LIN {X 0,Y 559.913,Z 737.575,A -85,B 0,C 180,E1 26462.456,E2 26462.456} C_VEL
LIN {X 0,Y 559.908,Z 738.885,A -85,B 0,C 180,E1 26460.511,E2 26460.511} C_VEL
LIN {X 0,Y 559.912,Z 738.467,A -85,B 0,C 180,E1 26458.465,E2 26458.465} C_VEL
LIN {X 0,Y 559.91,Z 736.338,A -85,B 0,C 180,E1 26456.519,E2 26456.519} C_VEL
LIN {X 0,Y 559.924,Z 732.455,A -85,B 0,C 180,E1 26454.569,E2 26454.569} C_VEL
LIN {X 0,Y 559.957,Z 726.723,A -85,B 0,C 180,E1 26452.613,E2 26452.613} C_VEL
LIN {X 0,Y 560.036,Z 718.997,A -85,B 0,C 180,E1 26450.649,E2 26450.649} C_VEL
LIN {X 0,Y 560.157,Z 709.621,A -85,B 0,C 180,E1 26448.781,E2 26448.781} C_VEL
LIN {X 0,Y 560.34,Z 698.616,A -85,B 0,C 180,E1 26447.007,E2 26447.007} C_VEL
LIN {X 0,Y 560.569,Z 686.811,A -85,B 0,C 180,E1 26445.434,E2 26445.434} C_VEL
LIN {X 0,Y 560.869,Z 673.245,A -85,B 0,C 180,E1 26443.921,E2 26443.921} C_VEL
LIN {X 0,Y 561.22,Z 658.578,A -85,B 0,C 180,E1 26442.549,E2 26442.549} C_VEL
LIN {X 0,Y 561.616,Z 642.337,A -85,B 0,C 180,E1 26441.287,E2 26441.287} C_VEL
LIN {X 0,Y 562.015,Z 624.834,A -85,B 0,C 180,E1 26440.178,E2 26440.178} C_VEL
LIN {X 0,Y 561.226,Z 618.186,A -85,B 0,C 180,E1 26439.775,E2 26439.775} C_VEL
LIN {X 0,Y 555.927,Z 601.44,A -85,B 0,C 180,E1 26438.77,E2 26438.77} C_VEL
LIN {X 0,Y 555.124,Z 594.384,A -85,B 0,C 180,E1 26438.452,E2 26438.452} C_VEL
LIN {X 0,Y 555.482,Z 575.161,A -85,B 0,C 180,E1 26437.832,E2 26437.832} C_VEL
LIN {X 0,Y 555.742,Z 555.75,A -85,B 0,C 180,E1 26437.414,E2 26437.414} C_VEL
LIN {X 0,Y 556.621,Z 349.619,A -85,B 0,C 180,E1 26434.588,E2 26434.588} C_VEL
LIN {X 0,Y 555.366,Z 342.045,A -85,B 0,C 180,E1 26434.399,E2 26434.399} C_VEL
LIN {X 0,Y 556.271,Z 299.379,A -85,B 0,C 180,E1 26431.026,E2 26431.026} C_VEL
LIN {X 0,Y 556.522,Z 280.46,A -85,B 0,C 180,E1 26429.484,E2 26429.484} C_VEL
LIN {X 0,Y 552.328,Z 267.902,A -85,B 0,C 180,E1 26428.132,E2 26428.132} C_VEL
LIN {X 0,Y 552.336,Z 267.663,A -85,B 0,C 180,E1 26425.089,E2 26425.089} C_VEL
LIN {X 0,Y 552.305,Z 267.685,A -85,B 0,C 180,E1 26421.746,E2 26421.746} C_VEL
LIN {X 0,Y 552.329,Z 267.679,A -85,B 0,C 180,E1 26418.366,E2 26418.366} C_VEL
LIN {X 0,Y 552.339,Z 267.686,A -85,B 0,C 180,E1 26415.057,E2 26415.057} C_VEL
LIN {X 0,Y 552.324,Z 267.684,A -85,B 0,C 180,E1 26411.768,E2 26411.768} C_VEL
LIN {X 0,Y 552.343,Z 267.678,A -85,B 0,C 180,E1 26408.383,E2 26408.383} C_VEL
LIN {X 0,Y 552.324,Z 267.683,A -85,B 0,C 180,E1 26405.02,E2 26405.02} C_VEL
LIN {X 0,Y 552.341,Z 267.686,A -85,B 0,C 180,E1 26401.667,E2 26401.667} C_VEL
LIN {X 0,Y 552.342,Z 267.677,A -85,B 0,C 180,E1 26398.313,E2 26398.313} C_VEL
LIN {X 0,Y 552.304,Z 267.68,A -85,B 0,C 180,E1 26394.95,E2 26394.95} C_VEL
LIN {X 0,Y 552.333,Z 267.683,A -85,B 0,C 180,E1 26391.673,E2 26391.673} C_VEL
LIN {X 0,Y 552.325,Z 267.683,A -85,B 0,C 180,E1 26388.361,E2 26388.361} C_VEL
LIN {X 0,Y 552.28,Z 267.68,A -85,B 0,C 180,E1 26385.113,E2 26385.113} C_VEL
LIN {X 0,Y 552.331,Z 267.688,A -85,B 0,C 180,E1 26381.911,E2 26381.911} C_VEL
LIN {X 0,Y 552.275,Z 267.688,A -85,B 0,C 180,E1 26378.695,E2 26378.695} C_VEL
LIN {X 0,Y 552.348,Z 268.019,A -85,B 0,C 180,E1 26378.406,E2 26378.406} C_VEL
LIN {X 0,Y 555.682,Z 279.748,A -85,B 0,C 180,E1 26377.289,E2 26377.289} C_VEL
LIN {X 0,Y 555.546,Z 319.159,A -85,B 0,C 180,E1 26374.233,E2 26374.233} C_VEL
LIN {X 0,Y 555.163,Z 359.793,A -85,B 0,C 180,E1 26371.085,E2 26371.085} C_VEL
LIN {X 0,Y 554.627,Z 395.794,A -85,B 0,C 180,E1 26368.297,E2 26368.297} C_VEL
LIN {X 0,Y 553.969,Z 440.023,A -85,B 0,C 180,E1 26364.875,E2 26364.875} C_VEL
LIN {X 0,Y 553.523,Z 472.352,A -85,B 0,C 180,E1 26362.411,E2 26362.411} C_VEL
LIN {X 0,Y 554.186,Z 480.588,A -85,B 0,C 180,E1 26362.264,E2 26362.264} C_VEL
LIN {X 0,Y 553.701,Z 615.423,A -85,B 0,C 180,E1 26360.465,E2 26360.465} C_VEL
LIN {X 0,Y 553.549,Z 631.717,A -85,B 0,C 180,E1 26360.048,E2 26360.048} C_VEL
LIN {X 0,Y 553.324,Z 647.903,A -85,B 0,C 180,E1 26359.427,E2 26359.427} C_VEL
LIN {X 0,Y 553.052,Z 662.877,A -85,B 0,C 180,E1 26358.636,E2 26358.636} C_VEL
LIN {X 0,Y 552.78,Z 676.977,A -85,B 0,C 180,E1 26357.678,E2 26357.678} C_VEL
LIN {X 0,Y 552.532,Z 689.984,A -85,B 0,C 180,E1 26356.555,E2 26356.555} C_VEL
LIN {X 0,Y 552.317,Z 701.515,A -85,B 0,C 180,E1 26355.32,E2 26355.32} C_VEL
LIN {X 0,Y 552.148,Z 711.975,A -85,B 0,C 180,E1 26353.917,E2 26353.917} C_VEL
LIN {X 0,Y 552.028,Z 720.937,A -85,B 0,C 180,E1 26352.395,E2 26352.395} C_VEL
LIN {X 0,Y 551.961,Z 727.845,A -85,B 0,C 180,E1 26350.862,E2 26350.862} C_VEL
LIN {X 0,Y 551.93,Z 733.356,A -85,B 0,C 180,E1 26349.192,E2 26349.192} C_VEL
LIN {X 0,Y 551.919,Z 736.92,A -85,B 0,C 180,E1 26347.529,E2 26347.529} C_VEL
LIN {X 0,Y 551.918,Z 738.738,A -85,B 0,C 180,E1 26345.833,E2 26345.833} C_VEL
LIN {X 0,Y 551.914,Z 738.822,A -85,B 0,C 180,E1 26344.209,E2 26344.209} C_VEL
LIN {X 0,Y 551.916,Z 737.077,A -85,B 0,C 180,E1 26342.488,E2 26342.488} C_VEL
LIN {X 0,Y 551.93,Z 733.669,A -85,B 0,C 180,E1 26340.831,E2 26340.831} C_VEL
LIN {X 0,Y 551.959,Z 728.277,A -85,B 0,C 180,E1 26339.161,E2 26339.161} C_VEL
LIN {X 0,Y 552.027,Z 721.222,A -85,B 0,C 180,E1 26337.571,E2 26337.571} C_VEL
LIN {X 0,Y 552.143,Z 712.252,A -85,B 0,C 180,E1 26336.036,E2 26336.036} C_VEL
LIN {X 0,Y 552.308,Z 702.136,A -85,B 0,C 180,E1 26334.664,E2 26334.664} C_VEL
LIN {X 0,Y 552.525,Z 690.435,A -85,B 0,C 180,E1 26333.399,E2 26333.399} C_VEL
LIN {X 0,Y 552.765,Z 678.003,A -85,B 0,C 180,E1 26332.312,E2 26332.312} C_VEL
LIN {X 0,Y 553.024,Z 664.254,A -85,B 0,C 180,E1 26331.358,E2 26331.358} C_VEL
LIN {X 0,Y 553.293,Z 649.215,A -85,B 0,C 180,E1 26330.544,E2 26330.544} C_VEL
LIN {X 0,Y 553.53,Z 633.394,A -85,B 0,C 180,E1 26329.917,E2 26329.917} C_VEL
LIN {X 0,Y 553.679,Z 617.007,A -85,B 0,C 180,E1 26329.476,E2 26329.476} C_VEL
LIN {X 0,Y 553.797,Z 584.698,A -85,B 0,C 180,E1 26329.014,E2 26329.014} C_VEL
LIN {X 0,Y 553.976,Z 476.401,A -85,B 0,C 180,E1 26327.584,E2 26327.584} C_VEL
LIN {X 0,Y 553.484,Z 472.041,A -85,B 0,C 180,E1 26327.481,E2 26327.481} C_VEL
LIN {X 0,Y 554.149,Z 429.88,A -85,B 0,C 180,E1 26324.252,E2 26324.252} C_VEL
LIN {X 0,Y 554.787,Z 388.2,A -85,B 0,C 180,E1 26320.997,E2 26320.997} C_VEL
LIN {X 0,Y 555.175,Z 355.136,A -85,B 0,C 180,E1 26318.48,E2 26318.48} C_VEL
LIN {X 0,Y 555.428,Z 312.632,A -85,B 0,C 180,E1 26315.231,E2 26315.231} C_VEL
LIN {X 0,Y 555.275,Z 277.84,A -85,B 0,C 180,E1 26312.575,E2 26312.575} C_VEL
LIN {X 0,Y 552.382,Z 267.955,A -85,B 0,C 180,E1 26311.648,E2 26311.648} C_VEL
LIN {X 0,Y 552.345,Z 267.684,A -85,B 0,C 180,E1 26309.463,E2 26309.463} C_VEL
LIN {X 0,Y 552.309,Z 267.688,A -85,B 0,C 180,E1 26306.118,E2 26306.118} C_VEL
LIN {X 0,Y 552.303,Z 267.684,A -85,B 0,C 180,E1 26302.794,E2 26302.794} C_VEL
LIN {X 0,Y 552.343,Z 267.684,A -85,B 0,C 180,E1 26299.566,E2 26299.566} C_VEL
LIN {X 0,Y 552.297,Z 267.686,A -85,B 0,C 180,E1 26296.297,E2 26296.297} C_VEL
LIN {X 0,Y 552.324,Z 267.681,A -85,B 0,C 180,E1 26292.972,E2 26292.972} C_VEL
LIN {X 0,Y 552.334,Z 267.688,A -85,B 0,C 180,E1 26289.692,E2 26289.692} C_VEL
LIN {X 0,Y 552.299,Z 267.683,A -85,B 0,C 180,E1 26286.356,E2 26286.356} C_VEL
LIN {X 0,Y 552.337,Z 267.681,A -85,B 0,C 180,E1 26283.01,E2 26283.01} C_VEL
LIN {X 0,Y 552.329,Z 267.687,A -85,B 0,C 180,E1 26279.689,E2 26279.689} C_VEL
LIN {X 0,Y 552.302,Z 267.682,A -85,B 0,C 180,E1 26276.368,E2 26276.368} C_VEL
LIN {X 0,Y 552.343,Z 267.68,A -85,B 0,C 180,E1 26273.034,E2 26273.034} C_VEL
LIN {X 0,Y 552.321,Z 267.685,A -85,B 0,C 180,E1 26269.676,E2 26269.676} C_VEL
LIN {X 0,Y 552.304,Z 267.682,A -85,B 0,C 180,E1 26266.282,E2 26266.282} C_VEL
LIN {X 0,Y 552.342,Z 267.682,A -85,B 0,C 180,E1 26263.056,E2 26263.056} C_VEL
LIN {X 0,Y 552.311,Z 267.685,A -85,B 0,C 180,E1 26259.771,E2 26259.771} C_VEL
LIN {X 0,Y 552.31,Z 267.682,A -85,B 0,C 180,E1 26256.304,E2 26256.304} C_VEL
LIN {X 0,Y 552.342,Z 267.682,A -85,B 0,C 180,E1 26252.976,E2 26252.976} C_VEL
LIN {X 0,Y 552.312,Z 267.684,A -85,B 0,C 180,E1 26249.664,E2 26249.664} C_VEL
LIN {X 0,Y 552.312,Z 267.681,A -85,B 0,C 180,E1 26246.192,E2 26246.192} C_VEL
LIN {X 0,Y 552.342,Z 267.683,A -85,B 0,C 180,E1 26242.929,E2 26242.929} C_VEL
LIN {X 0,Y 552.313,Z 267.685,A -85,B 0,C 180,E1 26239.602,E2 26239.602} C_VEL
LIN {X 0,Y 552.323,Z 267.682,A -85,B 0,C 180,E1 26236.242,E2 26236.242} C_VEL
LIN {X 0,Y 552.341,Z 267.685,A -85,B 0,C 180,E1 26232.892,E2 26232.892} C_VEL
LIN {X 0,Y 552.31,Z 267.686,A -85,B 0,C 180,E1 26229.584,E2 26229.584} C_VEL
LIN {X 0,Y 552.321,Z 267.656,A -85,B 0,C 180,E1 26226.166,E2 26226.166} C_VEL
LIN {X 0,Y 552.36,Z 267.887,A -85,B 0,C 180,E1 26224.227,E2 26224.227} C_VEL
LIN {X 0,Y 554.065,Z 272.818,A -85,B 0,C 180,E1 26223.704,E2 26223.704} C_VEL
LIN {X 0,Y 557.956,Z 283.115,A -85,B 0,C 180,E1 26222.701,E2 26222.701} C_VEL
LIN {X 0,Y 557.276,Z 315.739,A -85,B 0,C 180,E1 26220.45,E2 26220.45} C_VEL
LIN {X 0,Y 558.737,Z 325.763,A -85,B 0,C 180,E1 26220.212,E2 26220.212} C_VEL
LIN {X 0,Y 557.399,Z 554.976,A -85,B 0,C 180,E1 26216.995,E2 26216.995} C_VEL
LIN {X 0,Y 557.13,Z 582.184,A -85,B 0,C 180,E1 26216.559,E2 26216.559} C_VEL
LIN {X 0,Y 556.781,Z 602.596,A -85,B 0,C 180,E1 26216.039,E2 26216.039} C_VEL
LIN {X 0,Y 556.348,Z 622.128,A -85,B 0,C 180,E1 26215.354,E2 26215.354} C_VEL
LIN {X 0,Y 555.779,Z 641.891,A -85,B 0,C 180,E1 26214.453,E2 26214.453} C_VEL
LIN {X 0,Y 555.201,Z 660.724,A -85,B 0,C 180,E1 26213.385,E2 26213.385} C_VEL
LIN {X 0,Y 554.601,Z 678.942,A -85,B 0,C 180,E1 26212.134,E2 26212.134} C_VEL
LIN {X 0,Y 554.011,Z 696.238,A -85,B 0,C 180,E1 26210.714,E2 26210.714} C_VEL
LIN {X 0,Y 553.49,Z 711.936,A -85,B 0,C 180,E1 26209.193,E2 26209.193} C_VEL
LIN {X 0,Y 553.04,Z 726.218,A -85,B 0,C 180,E1 26207.572,E2 26207.572} C_VEL
LIN {X 0,Y 552.662,Z 739.872,A -85,B 0,C 180,E1 26205.745,E2 26205.745} C_VEL
LIN {X 0,Y 552.363,Z 751.931,A -85,B 0,C 180,E1 26203.823,E2 26203.823} C_VEL
LIN {X 0,Y 552.149,Z 762.4,A -85,B 0,C 180,E1 26201.806,E2 26201.806} C_VEL
LIN {X 0,Y 552.03,Z 770.879,A -85,B 0,C 180,E1 26199.801,E2 26199.801} C_VEL
LIN {X 0,Y 551.96,Z 777.902,A -85,B 0,C 180,E1 26197.702,E2 26197.702} C_VEL
LIN {X 0,Y 551.921,Z 783.145,A -85,B 0,C 180,E1 26195.613,E2 26195.613} C_VEL
LIN {X 0,Y 551.904,Z 786.711,A -85,B 0,C 180,E1 26193.53,E2 26193.53} C_VEL
LIN {X 0,Y 551.9,Z 788.575,A -85,B 0,C 180,E1 26191.452,E2 26191.452} C_VEL
LIN {X 0,Y 551.902,Z 788.873,A -85,B 0,C 180,E1 26189.376,E2 26189.376} C_VEL
LIN {X 0,Y 551.911,Z 787.504,A -85,B 0,C 180,E1 26187.195,E2 26187.195} C_VEL
LIN {X 0,Y 551.92,Z 784.578,A -85,B 0,C 180,E1 26185.115,E2 26185.115} C_VEL
LIN {X 0,Y 551.938,Z 779.972,A -85,B 0,C 180,E1 26183.028,E2 26183.028} C_VEL
LIN {X 0,Y 551.987,Z 773.909,A -85,B 0,C 180,E1 26181.037,E2 26181.037} C_VEL
LIN {X 0,Y 552.092,Z 765.953,A -85,B 0,C 180,E1 26178.986,E2 26178.986} C_VEL
LIN {X 0,Y 552.263,Z 756.56,A -85,B 0,C 180,E1 26177.026,E2 26177.026} C_VEL
LIN {X 0,Y 552.522,Z 745.371,A -85,B 0,C 180,E1 26175.091,E2 26175.091} C_VEL
LIN {X 0,Y 552.877,Z 732.126,A -85,B 0,C 180,E1 26173.18,E2 26173.18} C_VEL
LIN {X 0,Y 553.325,Z 717.313,A -85,B 0,C 180,E1 26171.382,E2 26171.382} C_VEL
LIN {X 0,Y 553.854,Z 701.041,A -85,B 0,C 180,E1 26169.719,E2 26169.719} C_VEL
LIN {X 0,Y 554.433,Z 683.855,A -85,B 0,C 180,E1 26168.24,E2 26168.24} C_VEL
LIN {X 0,Y 555.015,Z 666.503,A -85,B 0,C 180,E1 26166.987,E2 26166.987} C_VEL
LIN {X 0,Y 555.592,Z 648.265,A -85,B 0,C 180,E1 26165.888,E2 26165.888} C_VEL
LIN {X 0,Y 556.121,Z 629.25,A -85,B 0,C 180,E1 26164.949,E2 26164.949} C_VEL
LIN {X 0,Y 556.633,Z 609.344,A -85,B 0,C 180,E1 26164.176,E2 26164.176} C_VEL
LIN {X 0,Y 557.07,Z 588.839,A -85,B 0,C 180,E1 26163.585,E2 26163.585} C_VEL
LIN {X 0,Y 557.318,Z 567.71,A -85,B 0,C 180,E1 26163.184,E2 26163.184} C_VEL
LIN {X 0,Y 558.686,Z 334.299,A -85,B 0,C 180,E1 26159.909,E2 26159.909} C_VEL
LIN {X 0,Y 558.522,Z 323.011,A -85,B 0,C 180,E1 26159.735,E2 26159.735} C_VEL
LIN {X 0,Y 557.204,Z 314.837,A -85,B 0,C 180,E1 26159.51,E2 26159.51} C_VEL
LIN {X 0,Y 557.862,Z 282.456,A -85,B 0,C 180,E1 26157.245,E2 26157.245} C_VEL
LIN {X 0,Y 552.372,Z 267.996,A -85,B 0,C 180,E1 26155.833,E2 26155.833} C_VEL
LIN {X 0,Y 552.332,Z 267.687,A -85,B 0,C 180,E1 26154.853,E2 26154.853} C_VEL
LIN {X 0,Y 552.345,Z 267.684,A -85,B 0,C 180,E1 26151.445,E2 26151.445} C_VEL
LIN {X 0,Y 552.304,Z 267.686,A -85,B 0,C 180,E1 26148.224,E2 26148.224} C_VEL
LIN {X 0,Y 552.336,Z 267.688,A -85,B 0,C 180,E1 26144.909,E2 26144.909} C_VEL
LIN {X 0,Y 552.327,Z 267.683,A -85,B 0,C 180,E1 26141.613,E2 26141.613} C_VEL
LIN {X 0,Y 552.298,Z 267.688,A -85,B 0,C 180,E1 26138.381,E2 26138.381} C_VEL
LIN {X 0,Y 552.345,Z 267.686,A -85,B 0,C 180,E1 26135.093,E2 26135.093} C_VEL
LIN {X 0,Y 552.319,Z 267.821,A -85,B 0,C 180,E1 26131.819,E2 26131.819} C_VEL
LIN {X 0,Y 552.771,Z 269.52,A -85,B 0,C 180,E1 26131.575,E2 26131.575} C_VEL
LIN {X 0,Y 556.692,Z 281.727,A -85,B 0,C 180,E1 26130.311,E2 26130.311} C_VEL
LIN {X 0,Y 555.725,Z 323.491,A -85,B 0,C 180,E1 26126.962,E2 26126.962} C_VEL
LIN {X 0,Y 555.391,Z 342.331,A -85,B 0,C 180,E1 26125.498,E2 26125.498} C_VEL
LIN {X 0,Y 556.752,Z 351.91,A -85,B 0,C 180,E1 26125.284,E2 26125.284} C_VEL
LIN {X 0,Y 555.703,Z 559.825,A -85,B 0,C 180,E1 26122.426,E2 26122.426} C_VEL
LIN {X 0,Y 555.419,Z 579.56,A -85,B 0,C 180,E1 26121.955,E2 26121.955} C_VEL
LIN {X 0,Y 555.062,Z 598.233,A -85,B 0,C 180,E1 26121.31,E2 26121.31} C_VEL
LIN {X 0,Y 554.625,Z 616.494,A -85,B 0,C 180,E1 26120.471,E2 26120.471} C_VEL
LIN {X 0,Y 554.16,Z 634.188,A -85,B 0,C 180,E1 26119.444,E2 26119.444} C_VEL
LIN {X 0,Y 553.694,Z 650.84,A -85,B 0,C 180,E1 26118.253,E2 26118.253} C_VEL
LIN {X 0,Y 553.251,Z 666.265,A -85,B 0,C 180,E1 26116.915,E2 26116.915} C_VEL
LIN {X 0,Y 552.858,Z 680.646,A -85,B 0,C 180,E1 26115.417,E2 26115.417} C_VEL
LIN {X 0,Y 552.542,Z 693.493,A -85,B 0,C 180,E1 26113.819,E2 26113.819} C_VEL
LIN {X 0,Y 552.293,Z 704.824,A -85,B 0,C 180,E1 26112.122,E2 26112.122} C_VEL
LIN {X 0,Y 552.12,Z 714.658,A -85,B 0,C 180,E1 26110.328,E2 26110.328} C_VEL
LIN {X 0,Y 552.001,Z 722.972,A -85,B 0,C 180,E1 26108.436,E2 26108.436} C_VEL
LIN {X 0,Y 551.942,Z 729.719,A -85,B 0,C 180,E1 26106.448,E2 26106.448} C_VEL
LIN {X 0,Y 551.914,Z 734.549,A -85,B 0,C 180,E1 26104.467,E2 26104.467} C_VEL
LIN {X 0,Y 551.913,Z 737.578,A -85,B 0,C 180,E1 26102.492,E2 26102.492} C_VEL
LIN {X 0,Y 551.909,Z 738.886,A -85,B 0,C 180,E1 26100.519,E2 26100.519} C_VEL
LIN {X 0,Y 551.911,Z 738.468,A -85,B 0,C 180,E1 26098.442,E2 26098.442} C_VEL
LIN {X 0,Y 551.91,Z 736.34,A -85,B 0,C 180,E1 26096.468,E2 26096.468} C_VEL
LIN {X 0,Y 551.928,Z 732.456,A -85,B 0,C 180,E1 26094.49,E2 26094.49} C_VEL
LIN {X 0,Y 551.965,Z 726.721,A -85,B 0,C 180,E1 26092.505,E2 26092.505} C_VEL
LIN {X 0,Y 552.061,Z 718.994,A -85,B 0,C 180,E1 26090.513,E2 26090.513} C_VEL
LIN {X 0,Y 552.207,Z 709.621,A -85,B 0,C 180,E1 26088.617,E2 26088.617} C_VEL
LIN {X 0,Y 552.424,Z 698.615,A -85,B 0,C 180,E1 26086.817,E2 26086.817} C_VEL
LIN {X 0,Y 552.725,Z 685.961,A -85,B 0,C 180,E1 26085.115,E2 26085.115} C_VEL
LIN {X 0,Y 553.089,Z 672.079,A -85,B 0,C 180,E1 26083.565,E2 26083.565} C_VEL
LIN {X 0,Y 553.514,Z 657.117,A -85,B 0,C 180,E1 26082.17,E2 26082.17} C_VEL
LIN {X 0,Y 553.984,Z 640.418,A -85,B 0,C 180,E1 26080.885,E2 26080.885} C_VEL
LIN {X 0,Y 554.455,Z 623.149,A -85,B 0,C 180,E1 26079.797,E2 26079.797} C_VEL
LIN {X 0,Y 554.885,Z 606.004,A -85,B 0,C 180,E1 26078.931,E2 26078.931} C_VEL
LIN {X 0,Y 555.124,Z 594.384,A -85,B 0,C 180,E1 26078.452,E2 26078.452} C_VEL
LIN {X 0,Y 554.33,Z 587.206,A -85,B 0,C 180,E1 26078.154,E2 26078.154} C_VEL
LIN {X 0,Y 549.287,Z 570.234,A -85,B 0,C 180,E1 26077.439,E2 26077.439} C_VEL
LIN {X 0,Y 548.272,Z 562.843,A -85,B 0,C 180,E1 26077.225,E2 26077.225} C_VEL
LIN {X 0,Y 548.266,Z 561.759,A -85,B 0,C 180,E1 26077.202,E2 26077.202} C_VEL
LIN {X 0,Y 548.538,Z 526.374,A -85,B 0,C 180,E1 26076.678,E2 26076.678} C_VEL
LIN {X 0,Y 549.356,Z 350.631,A -85,B 0,C 180,E1 26074.242,E2 26074.242} C_VEL
LIN {X 0,Y 547.921,Z 342.045,A -85,B 0,C 180,E1 26074.026,E2 26074.026} C_VEL
LIN {X 0,Y 548.988,Z 299.37,A -85,B 0,C 180,E1 26070.604,E2 26070.604} C_VEL
LIN {X 0,Y 549.296,Z 283.514,A -85,B 0,C 180,E1 26069.297,E2 26069.297} C_VEL
LIN {X 0,Y 544.384,Z 268.893,A -85,B 0,C 180,E1 26067.691,E2 26067.691} C_VEL
LIN {X 0,Y 544.401,Z 268.658,A -85,B 0,C 180,E1 26064.652,E2 26064.652} C_VEL
LIN {X 0,Y 544.398,Z 268.676,A -85,B 0,C 180,E1 26061.222,E2 26061.222} C_VEL
LIN {X 0,Y 544.374,Z 268.67,A -85,B 0,C 180,E1 26057.901,E2 26057.901} C_VEL
LIN {X 0,Y 544.403,Z 268.669,A -85,B 0,C 180,E1 26054.552,E2 26054.552} C_VEL
LIN {X 0,Y 544.397,Z 268.674,A -85,B 0,C 180,E1 26051.111,E2 26051.111} C_VEL
LIN {X 0,Y 544.393,Z 268.674,A -85,B 0,C 180,E1 26047.706,E2 26047.706} C_VEL
LIN {X 0,Y 544.402,Z 268.668,A -85,B 0,C 180,E1 26044.26,E2 26044.26} C_VEL
LIN {X 0,Y 544.377,Z 268.67,A -85,B 0,C 180,E1 26040.935,E2 26040.935} C_VEL
LIN {X 0,Y 544.397,Z 268.677,A -85,B 0,C 180,E1 26037.571,E2 26037.571} C_VEL
LIN {X 0,Y 544.403,Z 268.666,A -85,B 0,C 180,E1 26034.178,E2 26034.178} C_VEL
LIN {X 0,Y 544.358,Z 268.671,A -85,B 0,C 180,E1 26030.876,E2 26030.876} C_VEL
LIN {X 0,Y 544.37,Z 268.677,A -85,B 0,C 180,E1 26027.532,E2 26027.532} C_VEL
LIN {X 0,Y 544.378,Z 268.661,A -85,B 0,C 180,E1 26024.357,E2 26024.357} C_VEL
LIN {X 0,Y 544.332,Z 268.675,A -85,B 0,C 180,E1 26021.121,E2 26021.121} C_VEL
LIN {X 0,Y 544.35,Z 268.818,A -85,B 0,C 180,E1 26018.809,E2 26018.809} C_VEL
LIN {X 0,Y 545.018,Z 271.044,A -85,B 0,C 180,E1 26018.547,E2 26018.547} C_VEL
LIN {X 0,Y 548.268,Z 282.133,A -85,B 0,C 180,E1 26017.493,E2 26017.493} C_VEL
LIN {X 0,Y 548.042,Z 321.72,A -85,B 0,C 180,E1 26014.396,E2 26014.396} C_VEL
LIN {X 0,Y 547.589,Z 362.631,A -85,B 0,C 180,E1 26011.204,E2 26011.204} C_VEL
LIN {X 0,Y 546.939,Z 404.882,A -85,B 0,C 180,E1 26007.906,E2 26007.906} C_VEL
LIN {X 0,Y 546.175,Z 447.44,A -85,B 0,C 180,E1 26004.591,E2 26004.591} C_VEL
LIN {X 0,Y 545.823,Z 472.822,A -85,B 0,C 180,E1 26002.65,E2 26002.65} C_VEL
LIN {X 0,Y 546.547,Z 481.441,A -85,B 0,C 180,E1 26002.502,E2 26002.502} C_VEL
LIN {X 0,Y 545.989,Z 615.312,A -85,B 0,C 180,E1 26000.691,E2 26000.691} C_VEL
LIN {X 0,Y 545.815,Z 631.31,A -85,B 0,C 180,E1 26000.281,E2 26000.281} C_VEL
LIN {X 0,Y 545.557,Z 647.511,A -85,B 0,C 180,E1 25999.654,E2 25999.654} C_VEL
LIN {X 0,Y 545.268,Z 661.83,A -85,B 0,C 180,E1 25998.9,E2 25998.9} C_VEL
LIN {X 0,Y 544.939,Z 676.127,A -85,B 0,C 180,E1 25997.928,E2 25997.928} C_VEL
LIN {X 0,Y 544.665,Z 688.782,A -85,B 0,C 180,E1 25996.844,E2 25996.844} C_VEL
LIN {X 0,Y 544.4,Z 700.969,A -85,B 0,C 180,E1 25995.537,E2 25995.537} C_VEL
LIN {X 0,Y 544.21,Z 710.834,A -85,B 0,C 180,E1 25994.223,E2 25994.223} C_VEL
LIN {X 0,Y 544.061,Z 720.003,A -85,B 0,C 180,E1 25992.681,E2 25992.681} C_VEL
LIN {X 0,Y 543.978,Z 727.166,A -85,B 0,C 180,E1 25991.127,E2 25991.127} C_VEL
LIN {X 0,Y 543.931,Z 732.813,A -85,B 0,C 180,E1 25989.447,E2 25989.447} C_VEL
LIN {X 0,Y 543.922,Z 736.644,A -85,B 0,C 180,E1 25987.75,E2 25987.75} C_VEL
LIN {X 0,Y 543.916,Z 738.634,A -85,B 0,C 180,E1 25986.011,E2 25986.011} C_VEL
LIN {X 0,Y 543.916,Z 738.853,A -85,B 0,C 180,E1 25984.258,E2 25984.258} C_VEL
LIN {X 0,Y 543.917,Z 737.184,A -85,B 0,C 180,E1 25982.524,E2 25982.524} C_VEL
LIN {X 0,Y 543.932,Z 733.808,A -85,B 0,C 180,E1 25980.828,E2 25980.828} C_VEL
LIN {X 0,Y 543.964,Z 728.552,A -85,B 0,C 180,E1 25979.149,E2 25979.149} C_VEL
LIN {X 0,Y 544.043,Z 721.506,A -85,B 0,C 180,E1 25977.519,E2 25977.519} C_VEL
LIN {X 0,Y 544.17,Z 713.158,A -85,B 0,C 180,E1 25976.045,E2 25976.045} C_VEL
LIN {X 0,Y 544.363,Z 702.783,A -85,B 0,C 180,E1 25974.593,E2 25974.593} C_VEL
LIN {X 0,Y 544.611,Z 691.264,A -85,B 0,C 180,E1 25973.311,E2 25973.311} C_VEL
LIN {X 0,Y 544.895,Z 678.555,A -85,B 0,C 180,E1 25972.171,E2 25972.171} C_VEL
LIN {X 0,Y 545.193,Z 665.066,A -85,B 0,C 180,E1 25971.209,E2 25971.209} C_VEL
LIN {X 0,Y 545.503,Z 649.951,A -85,B 0,C 180,E1 25970.37,E2 25970.37} C_VEL
LIN {X 0,Y 545.777,Z 634.463,A -85,B 0,C 180,E1 25969.734,E2 25969.734} C_VEL
LIN {X 0,Y 545.961,Z 617.574,A -85,B 0,C 180,E1 25969.264,E2 25969.264} C_VEL
LIN {X 0,Y 546.08,Z 591.808,A -85,B 0,C 180,E1 25968.878,E2 25968.878} C_VEL
LIN {X 0,Y 546.334,Z 477.199,A -85,B 0,C 180,E1 25967.344,E2 25967.344} C_VEL
LIN {X 0,Y 545.789,Z 472.587,A -85,B 0,C 180,E1 25967.245,E2 25967.245} C_VEL
LIN {X 0,Y 546.359,Z 437.042,A -85,B 0,C 180,E1 25964.5,E2 25964.5} C_VEL
LIN {X 0,Y 547.126,Z 394.245,A -85,B 0,C 180,E1 25961.14,E2 25961.14} C_VEL
LIN {X 0,Y 547.621,Z 354.566,A -85,B 0,C 180,E1 25958.107,E2 25958.107} C_VEL
LIN {X 0,Y 547.909,Z 314.541,A -85,B 0,C 180,E1 25955.025,E2 25955.025} C_VEL
LIN {X 0,Y 547.813,Z 280.315,A -85,B 0,C 180,E1 25952.391,E2 25952.391} C_VEL
LIN {X 0,Y 544.436,Z 268.93,A -85,B 0,C 180,E1 25951.315,E2 25951.315} C_VEL
LIN {X 0,Y 544.369,Z 268.677,A -85,B 0,C 180,E1 25948.164,E2 25948.164} C_VEL
LIN {X 0,Y 544.362,Z 268.675,A -85,B 0,C 180,E1 25944.758,E2 25944.758} C_VEL
LIN {X 0,Y 544.406,Z 268.671,A -85,B 0,C 180,E1 25941.438,E2 25941.438} C_VEL
LIN {X 0,Y 544.369,Z 268.673,A -85,B 0,C 180,E1 25938.084,E2 25938.084} C_VEL
LIN {X 0,Y 544.364,Z 268.671,A -85,B 0,C 180,E1 25934.683,E2 25934.683} C_VEL
LIN {X 0,Y 544.404,Z 268.673,A -85,B 0,C 180,E1 25931.441,E2 25931.441} C_VEL
LIN {X 0,Y 544.363,Z 268.674,A -85,B 0,C 180,E1 25928.12,E2 25928.12} C_VEL
LIN {X 0,Y 544.369,Z 268.671,A -85,B 0,C 180,E1 25924.636,E2 25924.636} C_VEL
LIN {X 0,Y 544.405,Z 268.674,A -85,B 0,C 180,E1 25921.369,E2 25921.369} C_VEL
LIN {X 0,Y 544.363,Z 268.672,A -85,B 0,C 180,E1 25918.106,E2 25918.106} C_VEL
LIN {X 0,Y 544.385,Z 268.67,A -85,B 0,C 180,E1 25914.731,E2 25914.731} C_VEL
LIN {X 0,Y 544.406,Z 268.673,A -85,B 0,C 180,E1 25911.339,E2 25911.339} C_VEL
LIN {X 0,Y 544.365,Z 268.673,A -85,B 0,C 180,E1 25908.021,E2 25908.021} C_VEL
LIN {X 0,Y 544.386,Z 268.668,A -85,B 0,C 180,E1 25904.627,E2 25904.627} C_VEL
LIN {X 0,Y 544.403,Z 268.673,A -85,B 0,C 180,E1 25901.252,E2 25901.252} C_VEL
LIN {X 0,Y 544.364,Z 268.672,A -85,B 0,C 180,E1 25897.995,E2 25897.995} C_VEL
LIN {X 0,Y 544.395,Z 268.669,A -85,B 0,C 180,E1 25894.635,E2 25894.635} C_VEL
LIN {X 0,Y 544.403,Z 268.675,A -85,B 0,C 180,E1 25891.237,E2 25891.237} C_VEL
LIN {X 0,Y 544.367,Z 268.672,A -85,B 0,C 180,E1 25887.94,E2 25887.94} C_VEL
LIN {X 0,Y 544.402,Z 268.668,A -85,B 0,C 180,E1 25884.63,E2 25884.63} C_VEL
LIN {X 0,Y 544.403,Z 268.676,A -85,B 0,C 180,E1 25881.224,E2 25881.224} C_VEL
LIN {X 0,Y 544.369,Z 268.673,A -85,B 0,C 180,E1 25877.902,E2 25877.902} C_VEL
LIN {X 0,Y 544.403,Z 268.669,A -85,B 0,C 180,E1 25874.552,E2 25874.552} C_VEL
LIN {X 0,Y 544.404,Z 268.675,A -85,B 0,C 180,E1 25871.108,E2 25871.108} C_VEL
LIN {X 0,Y 544.369,Z 268.676,A -85,B 0,C 180,E1 25867.834,E2 25867.834} C_VEL
LIN {X 0,Y 544.429,Z 268.872,A -85,B 0,C 180,E1 25864.701,E2 25864.701} C_VEL
LIN {X 0,Y 546.406,Z 274.424,A -85,B 0,C 180,E1 25864.104,E2 25864.104} C_VEL
LIN {X 0,Y 550.825,Z 286.317,A -85,B 0,C 180,E1 25862.937,E2 25862.937} C_VEL
LIN {X 0,Y 550.139,Z 315.757,A -85,B 0,C 180,E1 25860.887,E2 25860.887} C_VEL
LIN {X 0,Y 551.816,Z 326.941,A -85,B 0,C 180,E1 25860.614,E2 25860.614} C_VEL
LIN {X 0,Y 550.262,Z 556.513,A -85,B 0,C 180,E1 25857.352,E2 25857.352} C_VEL
LIN {X 0,Y 549.951,Z 582.995,A -85,B 0,C 180,E1 25856.916,E2 25856.916} C_VEL
LIN {X 0,Y 549.528,Z 603.787,A -85,B 0,C 180,E1 25856.369,E2 25856.369} C_VEL
LIN {X 0,Y 549.038,Z 622.887,A -85,B 0,C 180,E1 25855.683,E2 25855.683} C_VEL
LIN {X 0,Y 548.397,Z 642.486,A -85,B 0,C 180,E1 25854.774,E2 25854.774} C_VEL
LIN {X 0,Y 547.724,Z 661.447,A -85,B 0,C 180,E1 25853.677,E2 25853.677} C_VEL
LIN {X 0,Y 547.025,Z 679.674,A -85,B 0,C 180,E1 25852.4,E2 25852.4} C_VEL
LIN {X 0,Y 546.345,Z 696.844,A -85,B 0,C 180,E1 25850.963,E2 25850.963} C_VEL
LIN {X 0,Y 545.715,Z 713.203,A -85,B 0,C 180,E1 25849.338,E2 25849.338} C_VEL
LIN {X 0,Y 545.178,Z 727.917,A -85,B 0,C 180,E1 25847.613,E2 25847.613} C_VEL
LIN {X 0,Y 544.771,Z 740.579,A -85,B 0,C 180,E1 25845.869,E2 25845.869} C_VEL
LIN {X 0,Y 544.432,Z 752.54,A -85,B 0,C 180,E1 25843.92,E2 25843.92} C_VEL
LIN {X 0,Y 544.187,Z 762.914,A -85,B 0,C 180,E1 25841.874,E2 25841.874} C_VEL
LIN {X 0,Y 544.047,Z 771.283,A -85,B 0,C 180,E1 25839.84,E2 25839.84} C_VEL
LIN {X 0,Y 543.966,Z 778.205,A -85,B 0,C 180,E1 25837.71,E2 25837.71} C_VEL
LIN {X 0,Y 543.921,Z 783.351,A -85,B 0,C 180,E1 25835.59,E2 25835.59} C_VEL
LIN {X 0,Y 543.903,Z 786.829,A -85,B 0,C 180,E1 25833.477,E2 25833.477} C_VEL
LIN {X 0,Y 543.9,Z 788.642,A -85,B 0,C 180,E1 25831.368,E2 25831.368} C_VEL
LIN {X 0,Y 543.906,Z 788.851,A -85,B 0,C 180,E1 25829.262,E2 25829.262} C_VEL
LIN {X 0,Y 543.91,Z 787.393,A -85,B 0,C 180,E1 25827.048,E2 25827.048} C_VEL
LIN {X 0,Y 543.914,Z 784.373,A -85,B 0,C 180,E1 25824.937,E2 25824.937} C_VEL
LIN {X 0,Y 543.941,Z 779.709,A -85,B 0,C 180,E1 25822.818,E2 25822.818} C_VEL
LIN {X 0,Y 544.01,Z 773.367,A -85,B 0,C 180,E1 25820.741,E2 25820.741} C_VEL
LIN {X 0,Y 544.134,Z 765.716,A -85,B 0,C 180,E1 25818.767,E2 25818.767} C_VEL
LIN {X 0,Y 544.347,Z 755.986,A -85,B 0,C 180,E1 25816.725,E2 25816.725} C_VEL
LIN {X 0,Y 544.646,Z 744.783,A -85,B 0,C 180,E1 25814.779,E2 25814.779} C_VEL
LIN {X 0,Y 545.063,Z 731.768,A -85,B 0,C 180,E1 25812.885,E2 25812.885} C_VEL
LIN {X 0,Y 545.57,Z 717.476,A -85,B 0,C 180,E1 25811.126,E2 25811.126} C_VEL
LIN {X 0,Y 546.181,Z 701.37,A -85,B 0,C 180,E1 25809.453,E2 25809.453} C_VEL
LIN {X 0,Y 546.853,Z 684.004,A -85,B 0,C 180,E1 25807.935,E2 25807.935} C_VEL
LIN {X 0,Y 547.526,Z 666.499,A -85,B 0,C 180,E1 25806.654,E2 25806.654} C_VEL
LIN {X 0,Y 548.212,Z 647.865,A -85,B 0,C 180,E1 25805.519,E2 25805.519} C_VEL
LIN {X 0,Y 548.858,Z 627.964,A -85,B 0,C 180,E1 25804.536,E2 25804.536} C_VEL
LIN {X 0,Y 549.414,Z 607.739,A -85,B 0,C 180,E1 25803.757,E2 25803.757} C_VEL
LIN {X 0,Y 549.907,Z 587.593,A -85,B 0,C 180,E1 25803.185,E2 25803.185} C_VEL
LIN {X 0,Y 550.198,Z 566.503,A -85,B 0,C 180,E1 25802.788,E2 25802.788} C_VEL
LIN {X 0,Y 551.769,Z 333.79,A -85,B 0,C 180,E1 25799.485,E2 25799.485} C_VEL
LIN {X 0,Y 551.592,Z 324.232,A -85,B 0,C 180,E1 25799.332,E2 25799.332} C_VEL
LIN {X 0,Y 550.068,Z 315.089,A -85,B 0,C 180,E1 25799.087,E2 25799.087} C_VEL
LIN {X 0,Y 550.7,Z 285.522,A -85,B 0,C 180,E1 25797.015,E2 25797.015} C_VEL
LIN {X 0,Y 544.476,Z 269.148,A -85,B 0,C 180,E1 25795.427,E2 25795.427} C_VEL
LIN {X 0,Y 544.404,Z 268.675,A -85,B 0,C 180,E1 25794.997,E2 25794.997} C_VEL
LIN {X 0,Y 544.399,Z 268.673,A -85,B 0,C 180,E1 25791.626,E2 25791.626} C_VEL
LIN {X 0,Y 544.366,Z 268.676,A -85,B 0,C 180,E1 25788.325,E2 25788.325} C_VEL
LIN {X 0,Y 544.401,Z 268.676,A -85,B 0,C 180,E1 25784.999,E2 25784.999} C_VEL
LIN {X 0,Y 544.388,Z 268.673,A -85,B 0,C 180,E1 25781.623,E2 25781.623} C_VEL
LIN {X 0,Y 544.358,Z 268.677,A -85,B 0,C 180,E1 25778.343,E2 25778.343} C_VEL
LIN {X 0,Y 544.404,Z 268.676,A -85,B 0,C 180,E1 25775.001,E2 25775.001} C_VEL
LIN {X 0,Y 544.389,Z 268.94,A -85,B 0,C 180,E1 25772.245,E2 25772.245} C_VEL
LIN {X 0,Y 548.234,Z 280.298,A -85,B 0,C 180,E1 25770.951,E2 25770.951} C_VEL
LIN {X 0,Y 549.396,Z 284.616,A -85,B 0,C 180,E1 25770.514,E2 25770.514} C_VEL
LIN {X 0,Y 548.278,Z 326.381,A -85,B 0,C 180,E1 25767.123,E2 25767.123} C_VEL
LIN {X 0,Y 547.947,Z 342.348,A -85,B 0,C 180,E1 25765.87,E2 25765.87} C_VEL
LIN {X 0,Y 549.515,Z 352.978,A -85,B 0,C 180,E1 25765.627,E2 25765.627} C_VEL
LIN {X 0,Y 548.308,Z 559.851,A -85,B 0,C 180,E1 25762.746,E2 25762.746} C_VEL
LIN {X 0,Y 547.981,Z 579.575,A -85,B 0,C 180,E1 25762.268,E2 25762.268} C_VEL
LIN {X 0,Y 547.57,Z 598.25,A -85,B 0,C 180,E1 25761.616,E2 25761.616} C_VEL
LIN {X 0,Y 547.067,Z 616.503,A -85,B 0,C 180,E1 25760.767,E2 25760.767} C_VEL
LIN {X 0,Y 546.527,Z 634.25,A -85,B 0,C 180,E1 25759.723,E2 25759.723} C_VEL
LIN {X 0,Y 545.994,Z 650.785,A -85,B 0,C 180,E1 25758.525,E2 25758.525} C_VEL
LIN {X 0,Y 545.477,Z 666.271,A -85,B 0,C 180,E1 25757.164,E2 25757.164} C_VEL
LIN {X 0,Y 545.009,Z 681.023,A -85,B 0,C 180,E1 25755.601,E2 25755.601} C_VEL
LIN {X 0,Y 544.633,Z 694.276,A -85,B 0,C 180,E1 25753.915,E2 25753.915} C_VEL
LIN {X 0,Y 544.348,Z 705.47,A -85,B 0,C 180,E1 25752.194,E2 25752.194} C_VEL
LIN {X 0,Y 544.148,Z 715.181,A -85,B 0,C 180,E1 25750.374,E2 25750.374} C_VEL
LIN {X 0,Y 544.013,Z 723.379,A -85,B 0,C 180,E1 25748.455,E2 25748.455} C_VEL
LIN {X 0,Y 543.947,Z 730.024,A -85,B 0,C 180,E1 25746.438,E2 25746.438} C_VEL
LIN {X 0,Y 543.916,Z 734.758,A -85,B 0,C 180,E1 25744.428,E2 25744.428} C_VEL
LIN {X 0,Y 543.913,Z 737.693,A -85,B 0,C 180,E1 25742.423,E2 25742.423} C_VEL
LIN {X 0,Y 543.906,Z 738.908,A -85,B 0,C 180,E1 25740.421,E2 25740.421} C_VEL
LIN {X 0,Y 543.91,Z 738.4,A -85,B 0,C 180,E1 25738.314,E2 25738.314} C_VEL
LIN {X 0,Y 543.909,Z 736.184,A -85,B 0,C 180,E1 25736.311,E2 25736.311} C_VEL
LIN {X 0,Y 543.934,Z 732.204,A -85,B 0,C 180,E1 25734.303,E2 25734.303} C_VEL
LIN {X 0,Y 543.974,Z 726.72,A -85,B 0,C 180,E1 25732.395,E2 25732.395} C_VEL
LIN {X 0,Y 544.085,Z 718.991,A -85,B 0,C 180,E1 25730.373,E2 25730.373} C_VEL
LIN {X 0,Y 544.26,Z 709.62,A -85,B 0,C 180,E1 25728.448,E2 25728.448} C_VEL
LIN {X 0,Y 544.515,Z 698.615,A -85,B 0,C 180,E1 25726.622,E2 25726.622} C_VEL
LIN {X 0,Y 544.866,Z 685.958,A -85,B 0,C 180,E1 25724.895,E2 25724.895} C_VEL
LIN {X 0,Y 545.3,Z 671.961,A -85,B 0,C 180,E1 25723.312,E2 25723.312} C_VEL
LIN {X 0,Y 545.786,Z 657.173,A -85,B 0,C 180,E1 25721.915,E2 25721.915} C_VEL
LIN {X 0,Y 546.31,Z 641.073,A -85,B 0,C 180,E1 25720.654,E2 25720.654} C_VEL
LIN {X 0,Y 546.844,Z 624.073,A -85,B 0,C 180,E1 25719.559,E2 25719.559} C_VEL
LIN {X 0,Y 547.365,Z 605.986,A -85,B 0,C 180,E1 25718.628,E2 25718.628} C_VEL
LIN {X 0,Y 547.825,Z 587.15,A -85,B 0,C 180,E1 25717.883,E2 25717.883} C_VEL
LIN {X 0,Y 548.195,Z 567.733,A -85,B 0,C 180,E1 25717.328,E2 25717.328} C_VEL
LIN {X 0,Y 548.266,Z 561.759,A -85,B 0,C 180,E1 25717.202,E2 25717.202} C_VEL
LIN {X 0,Y 547.467,Z 554.222,A -85,B 0,C 180,E1 25717.025,E2 25717.025} C_VEL
LIN {X 0,Y 541.849,Z 534.391,A -85,B 0,C 180,E1 25716.484,E2 25716.484} C_VEL
LIN {X 0,Y 541.182,Z 527.864,A -85,B 0,C 180,E1 25716.364,E2 25716.364} C_VEL
LIN {X 0,Y 542.134,Z 351.748,A -85,B 0,C 180,E1 25713.89,E2 25713.89} C_VEL
LIN {X 0,Y 540.5,Z 342.045,A -85,B 0,C 180,E1 25713.642,E2 25713.642} C_VEL
LIN {X 0,Y 541.733,Z 299.305,A -85,B 0,C 180,E1 25710.166,E2 25710.166} C_VEL
LIN {X 0,Y 541.998,Z 286.28,A -85,B 0,C 180,E1 25709.073,E2 25709.073} C_VEL
LIN {X 0,Y 536.481,Z 269.937,A -85,B 0,C 180,E1 25707.247,E2 25707.247} C_VEL
LIN {X 0,Y 536.419,Z 269.631,A -85,B 0,C 180,E1 25705.613,E2 25705.613} C_VEL
LIN {X 0,Y 536.435,Z 269.661,A -85,B 0,C 180,E1 25702.177,E2 25702.177} C_VEL
LIN {X 0,Y 536.464,Z 269.659,A -85,B 0,C 180,E1 25698.849,E2 25698.849} C_VEL
LIN {X 0,Y 536.456,Z 269.662,A -85,B 0,C 180,E1 25695.397,E2 25695.397} C_VEL
LIN {X 0,Y 536.445,Z 269.661,A -85,B 0,C 180,E1 25691.953,E2 25691.953} C_VEL
LIN {X 0,Y 536.465,Z 269.657,A -85,B 0,C 180,E1 25688.5,E2 25688.5} C_VEL
LIN {X 0,Y 536.447,Z 269.661,A -85,B 0,C 180,E1 25685.035,E2 25685.035} C_VEL
LIN {X 0,Y 536.464,Z 269.665,A -85,B 0,C 180,E1 25681.583,E2 25681.583} C_VEL
LIN {X 0,Y 536.464,Z 269.656,A -85,B 0,C 180,E1 25678.135,E2 25678.135} C_VEL
LIN {X 0,Y 536.43,Z 269.656,A -85,B 0,C 180,E1 25674.796,E2 25674.796} C_VEL
LIN {X 0,Y 536.427,Z 269.661,A -85,B 0,C 180,E1 25671.314,E2 25671.314} C_VEL
LIN {X 0,Y 536.466,Z 269.659,A -85,B 0,C 180,E1 25668.023,E2 25668.023} C_VEL
LIN {X 0,Y 536.406,Z 269.656,A -85,B 0,C 180,E1 25664.796,E2 25664.796} C_VEL
LIN {X 0,Y 536.398,Z 269.665,A -85,B 0,C 180,E1 25661.288,E2 25661.288} C_VEL
LIN {X 0,Y 536.424,Z 269.919,A -85,B 0,C 180,E1 25659.144,E2 25659.144} C_VEL
LIN {X 0,Y 540.848,Z 284.151,A -85,B 0,C 180,E1 25657.733,E2 25657.733} C_VEL
LIN {X 0,Y 540.57,Z 322.999,A -85,B 0,C 180,E1 25654.669,E2 25654.669} C_VEL
LIN {X 0,Y 540.041,Z 364.148,A -85,B 0,C 180,E1 25651.433,E2 25651.433} C_VEL
LIN {X 0,Y 539.314,Z 406.637,A -85,B 0,C 180,E1 25648.089,E2 25648.089} C_VEL
LIN {X 0,Y 538.499,Z 448.804,A -85,B 0,C 180,E1 25644.781,E2 25644.781} C_VEL
LIN {X 0,Y 538.099,Z 472.579,A -85,B 0,C 180,E1 25642.93,E2 25642.93} C_VEL
LIN {X 0,Y 538.922,Z 482.051,A -85,B 0,C 180,E1 25642.752,E2 25642.752} C_VEL
LIN {X 0,Y 538.288,Z 615.431,A -85,B 0,C 180,E1 25640.92,E2 25640.92} C_VEL
LIN {X 0,Y 538.091,Z 631.37,A -85,B 0,C 180,E1 25640.506,E2 25640.506} C_VEL
LIN {X 0,Y 537.799,Z 647.272,A -85,B 0,C 180,E1 25639.882,E2 25639.882} C_VEL
LIN {X 0,Y 537.472,Z 661.659,A -85,B 0,C 180,E1 25639.117,E2 25639.117} C_VEL
LIN {X 0,Y 537.098,Z 675.993,A -85,B 0,C 180,E1 25638.131,E2 25638.131} C_VEL
LIN {X 0,Y 536.784,Z 688.686,A -85,B 0,C 180,E1 25637.031,E2 25637.031} C_VEL
LIN {X 0,Y 536.485,Z 700.671,A -85,B 0,C 180,E1 25635.73,E2 25635.73} C_VEL
LIN {X 0,Y 536.251,Z 711.135,A -85,B 0,C 180,E1 25634.316,E2 25634.316} C_VEL
LIN {X 0,Y 536.081,Z 720.309,A -85,B 0,C 180,E1 25632.737,E2 25632.737} C_VEL
LIN {X 0,Y 535.987,Z 727.339,A -85,B 0,C 180,E1 25631.174,E2 25631.174} C_VEL
LIN {X 0,Y 535.933,Z 732.938,A -85,B 0,C 180,E1 25629.469,E2 25629.469} C_VEL
LIN {X 0,Y 535.923,Z 736.713,A -85,B 0,C 180,E1 25627.746,E2 25627.746} C_VEL
LIN {X 0,Y 535.916,Z 738.649,A -85,B 0,C 180,E1 25626.003,E2 25626.003} C_VEL
LIN {X 0,Y 535.915,Z 738.847,A -85,B 0,C 180,E1 25624.235,E2 25624.235} C_VEL
LIN {X 0,Y 535.917,Z 737.114,A -85,B 0,C 180,E1 25622.441,E2 25622.441} C_VEL
LIN {X 0,Y 535.933,Z 733.748,A -85,B 0,C 180,E1 25620.74,E2 25620.74} C_VEL
LIN {X 0,Y 535.972,Z 728.722,A -85,B 0,C 180,E1 25619.109,E2 25619.109} C_VEL
LIN {X 0,Y 536.059,Z 721.789,A -85,B 0,C 180,E1 25617.467,E2 25617.467} C_VEL
LIN {X 0,Y 536.202,Z 713.635,A -85,B 0,C 180,E1 25615.987,E2 25615.987} C_VEL
LIN {X 0,Y 536.414,Z 703.594,A -85,B 0,C 180,E1 25614.544,E2 25614.544} C_VEL
LIN {X 0,Y 536.695,Z 692.234,A -85,B 0,C 180,E1 25613.235,E2 25613.235} C_VEL
LIN {X 0,Y 537.025,Z 679.185,A -85,B 0,C 180,E1 25612.034,E2 25612.034} C_VEL
LIN {X 0,Y 537.373,Z 665.506,A -85,B 0,C 180,E1 25611.033,E2 25611.033} C_VEL
LIN {X 0,Y 537.728,Z 650.25,A -85,B 0,C 180,E1 25610.17,E2 25610.17} C_VEL
LIN {X 0,Y 538.04,Z 634.911,A -85,B 0,C 180,E1 25609.524,E2 25609.524} C_VEL
LIN {X 0,Y 538.253,Z 618.059,A -85,B 0,C 180,E1 25609.043,E2 25609.043} C_VEL
LIN {X 0,Y 538.382,Z 595.599,A -85,B 0,C 180,E1 25608.693,E2 25608.693} C_VEL
LIN {X 0,Y 538.715,Z 478.039,A -85,B 0,C 180,E1 25607.096,E2 25607.096} C_VEL
LIN {X 0,Y 538.066,Z 472.24,A -85,B 0,C 180,E1 25606.954,E2 25606.954} C_VEL
LIN {X 0,Y 538.872,Z 429.115,A -85,B 0,C 180,E1 25603.586,E2 25603.586} C_VEL
LIN {X 0,Y 539.475,Z 395.429,A -85,B 0,C 180,E1 25600.926,E2 25600.926} C_VEL
LIN {X 0,Y 540.077,Z 355.837,A -85,B 0,C 180,E1 25597.859,E2 25597.859} C_VEL
LIN {X 0,Y 540.416,Z 313.922,A -85,B 0,C 180,E1 25594.612,E2 25594.612} C_VEL
LIN {X 0,Y 540.347,Z 282.76,A -85,B 0,C 180,E1 25592.203,E2 25592.203} C_VEL
LIN {X 0,Y 536.478,Z 269.981,A -85,B 0,C 180,E1 25590.986,E2 25590.986} C_VEL
LIN {X 0,Y 536.426,Z 269.667,A -85,B 0,C 180,E1 25590.216,E2 25590.216} C_VEL
LIN {X 0,Y 536.424,Z 269.664,A -85,B 0,C 180,E1 25586.774,E2 25586.774} C_VEL
LIN {X 0,Y 536.468,Z 269.661,A -85,B 0,C 180,E1 25583.39,E2 25583.39} C_VEL
LIN {X 0,Y 536.434,Z 269.664,A -85,B 0,C 180,E1 25580.054,E2 25580.054} C_VEL
LIN {X 0,Y 536.423,Z 269.663,A -85,B 0,C 180,E1 25576.658,E2 25576.658} C_VEL
LIN {X 0,Y 536.467,Z 269.661,A -85,B 0,C 180,E1 25573.363,E2 25573.363} C_VEL
LIN {X 0,Y 536.432,Z 269.664,A -85,B 0,C 180,E1 25569.983,E2 25569.983} C_VEL
LIN {X 0,Y 536.425,Z 269.66,A -85,B 0,C 180,E1 25566.529,E2 25566.529} C_VEL
LIN {X 0,Y 536.465,Z 269.66,A -85,B 0,C 180,E1 25563.206,E2 25563.206} C_VEL
LIN {X 0,Y 536.435,Z 269.664,A -85,B 0,C 180,E1 25559.894,E2 25559.894} C_VEL
LIN {X 0,Y 536.429,Z 269.659,A -85,B 0,C 180,E1 25556.474,E2 25556.474} C_VEL
LIN {X 0,Y 536.465,Z 269.66,A -85,B 0,C 180,E1 25553.15,E2 25553.15} C_VEL
LIN {X 0,Y 536.438,Z 269.662,A -85,B 0,C 180,E1 25549.768,E2 25549.768} C_VEL
LIN {X 0,Y 536.427,Z 269.66,A -85,B 0,C 180,E1 25546.307,E2 25546.307} C_VEL
LIN {X 0,Y 536.465,Z 269.659,A -85,B 0,C 180,E1 25542.958,E2 25542.958} C_VEL
LIN {X 0,Y 536.445,Z 269.664,A -85,B 0,C 180,E1 25539.602,E2 25539.602} C_VEL
LIN {X 0,Y 536.43,Z 269.66,A -85,B 0,C 180,E1 25536.227,E2 25536.227} C_VEL
LIN {X 0,Y 536.463,Z 269.658,A -85,B 0,C 180,E1 25532.83,E2 25532.83} C_VEL
LIN {X 0,Y 536.453,Z 269.663,A -85,B 0,C 180,E1 25529.415,E2 25529.415} C_VEL
LIN {X 0,Y 536.429,Z 269.661,A -85,B 0,C 180,E1 25526.002,E2 25526.002} C_VEL
LIN {X 0,Y 536.463,Z 269.657,A -85,B 0,C 180,E1 25522.584,E2 25522.584} C_VEL
LIN {X 0,Y 536.466,Z 269.664,A -85,B 0,C 180,E1 25519.142,E2 25519.142} C_VEL
LIN {X 0,Y 536.431,Z 269.663,A -85,B 0,C 180,E1 25515.805,E2 25515.805} C_VEL
LIN {X 0,Y 536.461,Z 269.66,A -85,B 0,C 180,E1 25512.428,E2 25512.428} C_VEL
LIN {X 0,Y 536.468,Z 269.663,A -85,B 0,C 180,E1 25508.996,E2 25508.996} C_VEL
LIN {X 0,Y 536.428,Z 269.624,A -85,B 0,C 180,E1 25505.643,E2 25505.643} C_VEL
LIN {X 0,Y 536.498,Z 269.951,A -85,B 0,C 180,E1 25505.175,E2 25505.175} C_VEL
LIN {X 0,Y 543.692,Z 289.122,A -85,B 0,C 180,E1 25503.202,E2 25503.202} C_VEL
LIN {X 0,Y 543.017,Z 315.812,A -85,B 0,C 180,E1 25501.33,E2 25501.33} C_VEL
LIN {X 0,Y 544.922,Z 328.267,A -85,B 0,C 180,E1 25501.024,E2 25501.024} C_VEL
LIN {X 0,Y 543.148,Z 557.81,A -85,B 0,C 180,E1 25497.722,E2 25497.722} C_VEL
LIN {X 0,Y 542.802,Z 583.319,A -85,B 0,C 180,E1 25497.292,E2 25497.292} C_VEL
LIN {X 0,Y 542.312,Z 604.435,A -85,B 0,C 180,E1 25496.726,E2 25496.726} C_VEL
LIN {X 0,Y 541.744,Z 623.594,A -85,B 0,C 180,E1 25496.022,E2 25496.022} C_VEL
LIN {X 0,Y 541.035,Z 643.066,A -85,B 0,C 180,E1 25495.104,E2 25495.104} C_VEL
LIN {X 0,Y 540.269,Z 661.99,A -85,B 0,C 180,E1 25493.989,E2 25493.989} C_VEL
LIN {X 0,Y 539.5,Z 679.409,A -85,B 0,C 180,E1 25492.75,E2 25492.75} C_VEL
LIN {X 0,Y 538.724,Z 696.568,A -85,B 0,C 180,E1 25491.299,E2 25491.299} C_VEL
LIN {X 0,Y 538.003,Z 712.948,A -85,B 0,C 180,E1 25489.655,E2 25489.655} C_VEL
LIN {X 0,Y 537.417,Z 727.069,A -85,B 0,C 180,E1 25487.988,E2 25487.988} C_VEL
LIN {X 0,Y 536.939,Z 739.874,A -85,B 0,C 180,E1 25486.218,E2 25486.218} C_VEL
LIN {X 0,Y 536.543,Z 751.928,A -85,B 0,C 180,E1 25484.239,E2 25484.239} C_VEL
LIN {X 0,Y 536.248,Z 762.399,A -85,B 0,C 180,E1 25482.162,E2 25482.162} C_VEL
LIN {X 0,Y 536.08,Z 770.877,A -85,B 0,C 180,E1 25480.096,E2 25480.096} C_VEL
LIN {X 0,Y 535.98,Z 777.902,A -85,B 0,C 180,E1 25477.933,E2 25477.933} C_VEL
LIN {X 0,Y 535.933,Z 783.144,A -85,B 0,C 180,E1 25475.781,E2 25475.781} C_VEL
LIN {X 0,Y 535.908,Z 786.711,A -85,B 0,C 180,E1 25473.636,E2 25473.636} C_VEL
LIN {X 0,Y 535.9,Z 788.575,A -85,B 0,C 180,E1 25471.496,E2 25471.496} C_VEL
LIN {X 0,Y 535.902,Z 788.873,A -85,B 0,C 180,E1 25469.357,E2 25469.357} C_VEL
LIN {X 0,Y 535.911,Z 787.505,A -85,B 0,C 180,E1 25467.111,E2 25467.111} C_VEL
LIN {X 0,Y 535.916,Z 784.579,A -85,B 0,C 180,E1 25464.968,E2 25464.968} C_VEL
LIN {X 0,Y 535.945,Z 779.971,A -85,B 0,C 180,E1 25462.818,E2 25462.818} C_VEL
LIN {X 0,Y 536.019,Z 773.909,A -85,B 0,C 180,E1 25460.768,E2 25460.768} C_VEL
LIN {X 0,Y 536.176,Z 765.716,A -85,B 0,C 180,E1 25458.598,E2 25458.598} C_VEL
LIN {X 0,Y 536.419,Z 755.985,A -85,B 0,C 180,E1 25456.526,E2 25456.526} C_VEL
LIN {X 0,Y 536.765,Z 744.782,A -85,B 0,C 180,E1 25454.55,E2 25454.55} C_VEL
LIN {X 0,Y 537.235,Z 732.125,A -85,B 0,C 180,E1 25452.675,E2 25452.675} C_VEL
LIN {X 0,Y 537.809,Z 717.951,A -85,B 0,C 180,E1 25450.9,E2 25450.9} C_VEL
LIN {X 0,Y 538.49,Z 702.162,A -85,B 0,C 180,E1 25449.227,E2 25449.227} C_VEL
LIN {X 0,Y 539.199,Z 685.938,A -85,B 0,C 180,E1 25447.772,E2 25447.772} C_VEL
LIN {X 0,Y 539.991,Z 668.119,A -85,B 0,C 180,E1 25446.424,E2 25446.424} C_VEL
LIN {X 0,Y 540.789,Z 649.161,A -85,B 0,C 180,E1 25445.236,E2 25445.236} C_VEL
LIN {X 0,Y 541.485,Z 630.527,A -85,B 0,C 180,E1 25444.282,E2 25444.282} C_VEL
LIN {X 0,Y 542.15,Z 610.603,A -85,B 0,C 180,E1 25443.476,E2 25443.476} C_VEL
LIN {X 0,Y 542.707,Z 589.933,A -85,B 0,C 180,E1 25442.859,E2 25442.859} C_VEL
LIN {X 0,Y 543.037,Z 569.316,A -85,B 0,C 180,E1 25442.447,E2 25442.447} C_VEL
LIN {X 0,Y 544.86,Z 336.081,A -85,B 0,C 180,E1 25439.09,E2 25439.09} C_VEL
LIN {X 0,Y 544.695,Z 325.466,A -85,B 0,C 180,E1 25438.92,E2 25438.92} C_VEL
LIN {X 0,Y 542.92,Z 315.066,A -85,B 0,C 180,E1 25438.646,E2 25438.646} C_VEL
LIN {X 0,Y 543.437,Z 288.327,A -85,B 0,C 180,E1 25436.777,E2 25436.777} C_VEL
LIN {X 0,Y 536.523,Z 270.066,A -85,B 0,C 180,E1 25434.954,E2 25434.954} C_VEL
LIN {X 0,Y 536.43,Z 269.668,A -85,B 0,C 180,E1 25434.309,E2 25434.309} C_VEL
LIN {X 0,Y 536.466,Z 269.664,A -85,B 0,C 180,E1 25430.952,E2 25430.952} C_VEL
LIN {X 0,Y 536.46,Z 269.662,A -85,B 0,C 180,E1 25427.567,E2 25427.567} C_VEL
LIN {X 0,Y 536.423,Z 269.665,A -85,B 0,C 180,E1 25424.195,E2 25424.195} C_VEL
LIN {X 0,Y 536.452,Z 269.666,A -85,B 0,C 180,E1 25420.824,E2 25420.824} C_VEL
LIN {X 0,Y 536.464,Z 269.663,A -85,B 0,C 180,E1 25417.416,E2 25417.416} C_VEL
LIN {X 0,Y 536.417,Z 269.669,A -85,B 0,C 180,E1 25414.128,E2 25414.128} C_VEL
LIN {X 0,Y 536.479,Z 269.923,A -85,B 0,C 180,E1 25412.753,E2 25412.753} C_VEL
LIN {X 0,Y 541.851,Z 285.756,A -85,B 0,C 180,E1 25410.901,E2 25410.901} C_VEL
LIN {X 0,Y 542.092,Z 288.262,A -85,B 0,C 180,E1 25410.663,E2 25410.663} C_VEL
LIN {X 0,Y 540.798,Z 330.21,A -85,B 0,C 180,E1 25407.213,E2 25407.213} C_VEL
LIN {X 0,Y 540.524,Z 342.365,A -85,B 0,C 180,E1 25406.252,E2 25406.252} C_VEL
LIN {X 0,Y 542.297,Z 354.174,A -85,B 0,C 180,E1 25405.976,E2 25405.976} C_VEL
LIN {X 0,Y 540.93,Z 559.878,A -85,B 0,C 180,E1 25403.074,E2 25403.074} C_VEL
LIN {X 0,Y 540.561,Z 579.589,A -85,B 0,C 180,E1 25402.591,E2 25402.591} C_VEL
LIN {X 0,Y 540.109,Z 597.611,A -85,B 0,C 180,E1 25401.957,E2 25401.957} C_VEL
LIN {X 0,Y 539.561,Z 615.488,A -85,B 0,C 180,E1 25401.126,E2 25401.126} C_VEL
LIN {X 0,Y 538.941,Z 633.351,A -85,B 0,C 180,E1 25400.073,E2 25400.073} C_VEL
LIN {X 0,Y 538.339,Z 650.126,A -85,B 0,C 180,E1 25398.854,E2 25398.854} C_VEL
LIN {X 0,Y 537.743,Z 665.732,A -85,B 0,C 180,E1 25397.473,E2 25397.473} C_VEL
LIN {X 0,Y 537.229,Z 679.731,A -85,B 0,C 180,E1 25395.988,E2 25395.988} C_VEL
LIN {X 0,Y 536.794,Z 692.735,A -85,B 0,C 180,E1 25394.343,E2 25394.343} C_VEL
LIN {X 0,Y 536.451,Z 704.2,A -85,B 0,C 180,E1 25392.595,E2 25392.595} C_VEL
LIN {X 0,Y 536.197,Z 714.521,A -85,B 0,C 180,E1 25390.668,E2 25390.668} C_VEL
LIN {X 0,Y 536.044,Z 722.975,A -85,B 0,C 180,E1 25388.689,E2 25388.689} C_VEL
LIN {X 0,Y 535.953,Z 729.726,A -85,B 0,C 180,E1 25386.642,E2 25386.642} C_VEL
LIN {X 0,Y 535.92,Z 734.557,A -85,B 0,C 180,E1 25384.601,E2 25384.601} C_VEL
LIN {X 0,Y 535.913,Z 737.584,A -85,B 0,C 180,E1 25382.566,E2 25382.566} C_VEL
LIN {X 0,Y 535.909,Z 738.883,A -85,B 0,C 180,E1 25380.534,E2 25380.534} C_VEL
LIN {X 0,Y 535.911,Z 738.47,A -85,B 0,C 180,E1 25378.396,E2 25378.396} C_VEL
LIN {X 0,Y 535.909,Z 736.343,A -85,B 0,C 180,E1 25376.363,E2 25376.363} C_VEL
LIN {X 0,Y 535.936,Z 732.458,A -85,B 0,C 180,E1 25374.325,E2 25374.325} C_VEL
LIN {X 0,Y 535.986,Z 726.718,A -85,B 0,C 180,E1 25372.281,E2 25372.281} C_VEL
LIN {X 0,Y 536.111,Z 718.986,A -85,B 0,C 180,E1 25370.228,E2 25370.228} C_VEL
LIN {X 0,Y 536.314,Z 709.616,A -85,B 0,C 180,E1 25368.275,E2 25368.275} C_VEL
LIN {X 0,Y 536.612,Z 698.614,A -85,B 0,C 180,E1 25366.421,E2 25366.421} C_VEL
LIN {X 0,Y 537.018,Z 685.955,A -85,B 0,C 180,E1 25364.669,E2 25364.669} C_VEL
LIN {X 0,Y 537.514,Z 672.061,A -85,B 0,C 180,E1 25363.075,E2 25363.075} C_VEL
LIN {X 0,Y 538.075,Z 657.098,A -85,B 0,C 180,E1 25361.641,E2 25361.641} C_VEL
LIN {X 0,Y 538.673,Z 641.059,A -85,B 0,C 180,E1 25360.368,E2 25360.368} C_VEL
LIN {X 0,Y 539.277,Z 624.057,A -85,B 0,C 180,E1 25359.259,E2 25359.259} C_VEL
LIN {X 0,Y 539.834,Z 607.194,A -85,B 0,C 180,E1 25358.371,E2 25358.371} C_VEL
LIN {X 0,Y 540.353,Z 588.542,A -85,B 0,C 180,E1 25357.611,E2 25357.611} C_VEL
LIN {X 0,Y 540.775,Z 568.878,A -85,B 0,C 180,E1 25357.03,E2 25357.03} C_VEL
LIN {X 0,Y 541.052,Z 549.078,A -85,B 0,C 180,E1 25356.659,E2 25356.659} C_VEL
LIN {X 0,Y 541.182,Z 527.864,A -85,B 0,C 180,E1 25356.364,E2 25356.364} C_VEL
LIN {X 0,Y 540.307,Z 520.275,A -85,B 0,C 180,E1 25356.216,E2 25356.216} C_VEL
LIN {X 0,Y 534.727,Z 500.431,A -85,B 0,C 180,E1 25355.666,E2 25355.666} C_VEL
LIN {X 0,Y 534.074,Z 493.908,A -85,B 0,C 180,E1 25355.54,E2 25355.54} C_VEL
LIN {X 0,Y 534.906,Z 352.739,A -85,B 0,C 180,E1 25353.525,E2 25353.525} C_VEL
LIN {X 0,Y 533.102,Z 342.045,A -85,B 0,C 180,E1 25353.247,E2 25353.247} C_VEL
LIN {X 0,Y 534.497,Z 300.157,A -85,B 0,C 180,E1 25349.787,E2 25349.787} C_VEL
LIN {X 0,Y 534.882,Z 289.528,A -85,B 0,C 180,E1 25348.887,E2 25348.887} C_VEL
LIN {X 0,Y 528.554,Z 270.846,A -85,B 0,C 180,E1 25346.746,E2 25346.746} C_VEL
LIN {X 0,Y 528.493,Z 270.654,A -85,B 0,C 180,E1 25343.52,E2 25343.52} C_VEL
LIN {X 0,Y 528.494,Z 270.65,A -85,B 0,C 180,E1 25340.017,E2 25340.017} C_VEL
LIN {X 0,Y 528.526,Z 270.647,A -85,B 0,C 180,E1 25336.59,E2 25336.59} C_VEL
LIN {X 0,Y 528.52,Z 270.65,A -85,B 0,C 180,E1 25333.075,E2 25333.075} C_VEL
LIN {X 0,Y 528.516,Z 270.653,A -85,B 0,C 180,E1 25329.648,E2 25329.648} C_VEL
LIN {X 0,Y 528.516,Z 270.647,A -85,B 0,C 180,E1 25326.117,E2 25326.117} C_VEL
LIN {X 0,Y 528.507,Z 270.648,A -85,B 0,C 180,E1 25322.757,E2 25322.757} C_VEL
LIN {X 0,Y 528.503,Z 270.647,A -85,B 0,C 180,E1 25319.217,E2 25319.217} C_VEL
LIN {X 0,Y 528.526,Z 270.648,A -85,B 0,C 180,E1 25315.776,E2 25315.776} C_VEL
LIN {X 0,Y 528.519,Z 270.649,A -85,B 0,C 180,E1 25312.316,E2 25312.316} C_VEL
LIN {X 0,Y 528.476,Z 270.652,A -85,B 0,C 180,E1 25308.916,E2 25308.916} C_VEL
LIN {X 0,Y 528.481,Z 270.646,A -85,B 0,C 180,E1 25305.473,E2 25305.473} C_VEL
LIN {X 0,Y 528.509,Z 270.651,A -85,B 0,C 180,E1 25302.234,E2 25302.234} C_VEL
LIN {X 0,Y 528.497,Z 270.87,A -85,B 0,C 180,E1 25299.53,E2 25299.53} C_VEL
LIN {X 0,Y 533.456,Z 286.886,A -85,B 0,C 180,E1 25297.919,E2 25297.919} C_VEL
LIN {X 0,Y 533.075,Z 326.99,A -85,B 0,C 180,E1 25294.735,E2 25294.735} C_VEL
LIN {X 0,Y 532.459,Z 368.362,A -85,B 0,C 180,E1 25291.454,E2 25291.454} C_VEL
LIN {X 0,Y 531.647,Z 411.901,A -85,B 0,C 180,E1 25288.007,E2 25288.007} C_VEL
LIN {X 0,Y 530.729,Z 455.611,A -85,B 0,C 180,E1 25284.542,E2 25284.542} C_VEL
LIN {X 0,Y 530.457,Z 473.352,A -85,B 0,C 180,E1 25283.178,E2 25283.178} C_VEL
LIN {X 0,Y 531.307,Z 482.893,A -85,B 0,C 180,E1 25283.006,E2 25283.006} C_VEL
LIN {X 0,Y 530.599,Z 615.85,A -85,B 0,C 180,E1 25281.153,E2 25281.153} C_VEL
LIN {X 0,Y 530.385,Z 631.772,A -85,B 0,C 180,E1 25280.733,E2 25280.733} C_VEL
LIN {X 0,Y 530.074,Z 647.293,A -85,B 0,C 180,E1 25280.118,E2 25280.118} C_VEL
LIN {X 0,Y 529.71,Z 661.751,A -85,B 0,C 180,E1 25279.341,E2 25279.341} C_VEL
LIN {X 0,Y 529.286,Z 676.065,A -85,B 0,C 180,E1 25278.34,E2 25278.34} C_VEL
LIN {X 0,Y 528.924,Z 688.726,A -85,B 0,C 180,E1 25277.223,E2 25277.223} C_VEL
LIN {X 0,Y 528.567,Z 700.857,A -85,B 0,C 180,E1 25275.877,E2 25275.877} C_VEL
LIN {X 0,Y 528.292,Z 711.425,A -85,B 0,C 180,E1 25274.411,E2 25274.411} C_VEL
LIN {X 0,Y 528.102,Z 720.477,A -85,B 0,C 180,E1 25272.823,E2 25272.823} C_VEL
LIN {X 0,Y 527.995,Z 727.509,A -85,B 0,C 180,E1 25271.222,E2 25271.222} C_VEL
LIN {X 0,Y 527.936,Z 733.064,A -85,B 0,C 180,E1 25269.491,E2 25269.491} C_VEL
LIN {X 0,Y 527.923,Z 736.631,A -85,B 0,C 180,E1 25267.842,E2 25267.842} C_VEL
LIN {X 0,Y 527.916,Z 738.604,A -85,B 0,C 180,E1 25266.091,E2 25266.091} C_VEL
LIN {X 0,Y 527.915,Z 738.87,A -85,B 0,C 180,E1 25264.298,E2 25264.298} C_VEL
LIN {X 0,Y 527.917,Z 737.398,A -85,B 0,C 180,E1 25262.599,E2 25262.599} C_VEL
LIN {X 0,Y 527.935,Z 733.922,A -85,B 0,C 180,E1 25260.751,E2 25260.751} C_VEL
LIN {X 0,Y 527.978,Z 728.938,A -85,B 0,C 180,E1 25259.079,E2 25259.079} C_VEL
LIN {X 0,Y 528.083,Z 721.748,A -85,B 0,C 180,E1 25257.345,E2 25257.345} C_VEL
LIN {X 0,Y 528.251,Z 713.297,A -85,B 0,C 180,E1 25255.797,E2 25255.797} C_VEL
LIN {X 0,Y 528.524,Z 702.456,A -85,B 0,C 180,E1 25254.23,E2 25254.23} C_VEL
LIN {X 0,Y 528.854,Z 690.914,A -85,B 0,C 180,E1 25252.909,E2 25252.909} C_VEL
LIN {X 0,Y 529.242,Z 677.872,A -85,B 0,C 180,E1 25251.71,E2 25251.71} C_VEL
LIN {X 0,Y 529.638,Z 664.081,A -85,B 0,C 180,E1 25250.716,E2 25250.716} C_VEL
LIN {X 0,Y 530.042,Z 648.995,A -85,B 0,C 180,E1 25249.869,E2 25249.869} C_VEL
LIN {X 0,Y 530.364,Z 632.881,A -85,B 0,C 180,E1 25249.214,E2 25249.214} C_VEL
LIN {X 0,Y 530.581,Z 616.78,A -85,B 0,C 180,E1 25248.773,E2 25248.773} C_VEL
LIN {X 0,Y 530.833,Z 568.061,A -85,B 0,C 180,E1 25248.072,E2 25248.072} C_VEL
LIN {X 0,Y 531.109,Z 478.885,A -85,B 0,C 180,E1 25246.841,E2 25246.841} C_VEL
LIN {X 0,Y 530.394,Z 472.628,A -85,B 0,C 180,E1 25246.691,E2 25246.691} C_VEL
LIN {X 0,Y 531.251,Z 429.763,A -85,B 0,C 180,E1 25243.316,E2 25243.316} C_VEL
LIN {X 0,Y 532.007,Z 389.605,A -85,B 0,C 180,E1 25240.139,E2 25240.139} C_VEL
LIN {X 0,Y 532.616,Z 350.06,A -85,B 0,C 180,E1 25237.057,E2 25237.057} C_VEL
LIN {X 0,Y 532.94,Z 312.405,A -85,B 0,C 180,E1 25234.123,E2 25234.123} C_VEL
LIN {X 0,Y 532.852,Z 285.087,A -85,B 0,C 180,E1 25231.993,E2 25231.993} C_VEL
LIN {X 0,Y 528.518,Z 270.929,A -85,B 0,C 180,E1 25230.623,E2 25230.623} C_VEL
LIN {X 0,Y 528.488,Z 270.655,A -85,B 0,C 180,E1 25228.229,E2 25228.229} C_VEL
LIN {X 0,Y 528.484,Z 270.653,A -85,B 0,C 180,E1 25224.716,E2 25224.716} C_VEL
LIN {X 0,Y 528.528,Z 270.648,A -85,B 0,C 180,E1 25221.415,E2 25221.415} C_VEL
LIN {X 0,Y 528.492,Z 270.65,A -85,B 0,C 180,E1 25218.076,E2 25218.076} C_VEL
LIN {X 0,Y 528.488,Z 270.649,A -85,B 0,C 180,E1 25214.686,E2 25214.686} C_VEL
LIN {X 0,Y 528.527,Z 270.65,A -85,B 0,C 180,E1 25211.347,E2 25211.347} C_VEL
LIN {X 0,Y 528.496,Z 270.652,A -85,B 0,C 180,E1 25207.939,E2 25207.939} C_VEL
LIN {X 0,Y 528.488,Z 270.649,A -85,B 0,C 180,E1 25204.558,E2 25204.558} C_VEL
LIN {X 0,Y 528.527,Z 270.649,A -85,B 0,C 180,E1 25201.193,E2 25201.193} C_VEL
LIN {X 0,Y 528.499,Z 270.652,A -85,B 0,C 180,E1 25197.832,E2 25197.832} C_VEL
LIN {X 0,Y 528.486,Z 270.65,A -85,B 0,C 180,E1 25194.354,E2 25194.354} C_VEL
LIN {X 0,Y 528.527,Z 270.646,A -85,B 0,C 180,E1 25191.076,E2 25191.076} C_VEL
LIN {X 0,Y 528.506,Z 270.653,A -85,B 0,C 180,E1 25187.656,E2 25187.656} C_VEL
LIN {X 0,Y 528.49,Z 270.647,A -85,B 0,C 180,E1 25184.304,E2 25184.304} C_VEL
LIN {X 0,Y 528.526,Z 270.647,A -85,B 0,C 180,E1 25180.897,E2 25180.897} C_VEL
LIN {X 0,Y 528.519,Z 270.651,A -85,B 0,C 180,E1 25177.416,E2 25177.416} C_VEL
LIN {X 0,Y 528.489,Z 270.651,A -85,B 0,C 180,E1 25173.978,E2 25173.978} C_VEL
LIN {X 0,Y 528.514,Z 270.645,A -85,B 0,C 180,E1 25170.536,E2 25170.536} C_VEL
LIN {X 0,Y 528.526,Z 270.652,A -85,B 0,C 180,E1 25167.116,E2 25167.116} C_VEL
LIN {X 0,Y 528.494,Z 270.652,A -85,B 0,C 180,E1 25163.69,E2 25163.69} C_VEL
LIN {X 0,Y 528.5,Z 270.648,A -85,B 0,C 180,E1 25160.181,E2 25160.181} C_VEL
LIN {X 0,Y 528.526,Z 270.651,A -85,B 0,C 180,E1 25156.778,E2 25156.778} C_VEL
LIN {X 0,Y 528.509,Z 270.654,A -85,B 0,C 180,E1 25153.37,E2 25153.37} C_VEL
LIN {X 0,Y 528.496,Z 270.651,A -85,B 0,C 180,E1 25149.985,E2 25149.985} C_VEL
LIN {X 0,Y 528.519,Z 270.616,A -85,B 0,C 180,E1 25146.667,E2 25146.667} C_VEL
LIN {X 0,Y 528.529,Z 270.894,A -85,B 0,C 180,E1 25145.703,E2 25145.703} C_VEL
LIN {X 0,Y 530.564,Z 276.356,A -85,B 0,C 180,E1 25145.082,E2 25145.082} C_VEL
LIN {X 0,Y 536.57,Z 291.928,A -85,B 0,C 180,E1 25143.473,E2 25143.473} C_VEL
LIN {X 0,Y 535.869,Z 316.027,A -85,B 0,C 180,E1 25141.761,E2 25141.761} C_VEL
LIN {X 0,Y 537.956,Z 329.446,A -85,B 0,C 180,E1 25141.428,E2 25141.428} C_VEL
LIN {X 0,Y 536.141,Z 549.123,A -85,B 0,C 180,E1 25138.246,E2 25138.246} C_VEL
LIN {X 0,Y 535.77,Z 580.397,A -85,B 0,C 180,E1 25137.749,E2 25137.749} C_VEL
LIN {X 0,Y 535.266,Z 600.963,A -85,B 0,C 180,E1 25137.226,E2 25137.226} C_VEL
LIN {X 0,Y 534.596,Z 620.781,A -85,B 0,C 180,E1 25136.52,E2 25136.52} C_VEL
LIN {X 0,Y 533.837,Z 639.893,A -85,B 0,C 180,E1 25135.634,E2 25135.634} C_VEL
LIN {X 0,Y 532.985,Z 658.752,A -85,B 0,C 180,E1 25134.551,E2 25134.551} C_VEL
LIN {X 0,Y 532.069,Z 677.587,A -85,B 0,C 180,E1 25133.231,E2 25133.231} C_VEL
LIN {X 0,Y 531.234,Z 694.408,A -85,B 0,C 180,E1 25131.82,E2 25131.82} C_VEL
LIN {X 0,Y 530.443,Z 710.413,A -85,B 0,C 180,E1 25130.234,E2 25130.234} C_VEL
LIN {X 0,Y 529.729,Z 725.368,A -85,B 0,C 180,E1 25128.486,E2 25128.486} C_VEL
LIN {X 0,Y 529.125,Z 739.131,A -85,B 0,C 180,E1 25126.577,E2 25126.577} C_VEL
LIN {X 0,Y 528.68,Z 750.657,A -85,B 0,C 180,E1 25124.679,E2 25124.679} C_VEL
LIN {X 0,Y 528.348,Z 760.855,A -85,B 0,C 180,E1 25122.68,E2 25122.68} C_VEL
LIN {X 0,Y 528.124,Z 770.067,A -85,B 0,C 180,E1 25120.47,E2 25120.47} C_VEL
LIN {X 0,Y 528.002,Z 777.295,A -85,B 0,C 180,E1 25118.273,E2 25118.273} C_VEL
LIN {X 0,Y 527.944,Z 782.73,A -85,B 0,C 180,E1 25116.087,E2 25116.087} C_VEL
LIN {X 0,Y 527.918,Z 786.404,A -85,B 0,C 180,E1 25113.908,E2 25113.908} C_VEL
LIN {X 0,Y 527.906,Z 788.443,A -85,B 0,C 180,E1 25111.735,E2 25111.735} C_VEL
LIN {X 0,Y 527.9,Z 788.895,A -85,B 0,C 180,E1 25109.456,E2 25109.456} C_VEL
LIN {X 0,Y 527.911,Z 787.729,A -85,B 0,C 180,E1 25107.285,E2 25107.285} C_VEL
LIN {X 0,Y 527.922,Z 784.968,A -85,B 0,C 180,E1 25105.11,E2 25105.11} C_VEL
LIN {X 0,Y 527.948,Z 780.464,A -85,B 0,C 180,E1 25102.921,E2 25102.921} C_VEL
LIN {X 0,Y 528.031,Z 774.263,A -85,B 0,C 180,E1 25100.737,E2 25100.737} C_VEL
LIN {X 0,Y 528.207,Z 766.173,A -85,B 0,C 180,E1 25098.535,E2 25098.535} C_VEL
LIN {X 0,Y 528.478,Z 756.557,A -85,B 0,C 180,E1 25096.431,E2 25096.431} C_VEL
LIN {X 0,Y 528.869,Z 745.481,A -85,B 0,C 180,E1 25094.426,E2 25094.426} C_VEL
LIN {X 0,Y 529.395,Z 732.863,A -85,B 0,C 180,E1 25092.512,E2 25092.512} C_VEL
LIN {X 0,Y 530.029,Z 718.878,A -85,B 0,C 180,E1 25090.723,E2 25090.723} C_VEL
LIN {X 0,Y 530.753,Z 703.881,A -85,B 0,C 180,E1 25089.089,E2 25089.089} C_VEL
LIN {X 0,Y 531.581,Z 687.27,A -85,B 0,C 180,E1 25087.552,E2 25087.552} C_VEL
LIN {X 0,Y 532.465,Z 669.74,A -85,B 0,C 180,E1 25086.188,E2 25086.188} C_VEL
LIN {X 0,Y 533.347,Z 651.268,A -85,B 0,C 180,E1 25084.991,E2 25084.991} C_VEL
LIN {X 0,Y 534.152,Z 632.343,A -85,B 0,C 180,E1 25083.987,E2 25083.987} C_VEL
LIN {X 0,Y 534.891,Z 612.583,A -85,B 0,C 180,E1 25083.164,E2 25083.164} C_VEL
LIN {X 0,Y 535.481,Z 592.698,A -85,B 0,C 180,E1 25082.542,E2 25082.542} C_VEL
LIN {X 0,Y 535.906,Z 571.719,A -85,B 0,C 180,E1 25082.091,E2 25082.091} C_VEL
LIN {X 0,Y 537.478,Z 381.035,A -85,B 0,C 180,E1 25079.337,E2 25079.337} C_VEL
LIN {X 0,Y 537.602,Z 326.941,A -85,B 0,C 180,E1 25078.555,E2 25078.555} C_VEL
LIN {X 0,Y 535.65,Z 315.573,A -85,B 0,C 180,E1 25078.266,E2 25078.266} C_VEL
LIN {X 0,Y 536.239,Z 291.369,A -85,B 0,C 180,E1 25076.553,E2 25076.553} C_VEL
LIN {X 0,Y 528.555,Z 271.061,A -85,B 0,C 180,E1 25074.464,E2 25074.464} C_VEL
LIN {X 0,Y 528.509,Z 270.655,A -85,B 0,C 180,E1 25073.824,E2 25073.824} C_VEL
LIN {X 0,Y 528.489,Z 270.655,A -85,B 0,C 180,E1 25070.354,E2 25070.354} C_VEL
LIN {X 0,Y 528.525,Z 270.653,A -85,B 0,C 180,E1 25067.064,E2 25067.064} C_VEL
LIN {X 0,Y 528.508,Z 270.652,A -85,B 0,C 180,E1 25063.671,E2 25063.671} C_VEL
LIN {X 0,Y 528.483,Z 270.656,A -85,B 0,C 180,E1 25060.318,E2 25060.318} C_VEL
LIN {X 0,Y 528.522,Z 270.654,A -85,B 0,C 180,E1 25056.984,E2 25056.984} C_VEL
LIN {X 0,Y 528.499,Z 270.655,A -85,B 0,C 180,E1 25053.65,E2 25053.65} C_VEL
LIN {X 0,Y 528.597,Z 271.112,A -85,B 0,C 180,E1 25053.256,E2 25053.256} C_VEL
LIN {X 0,Y 534.257,Z 287.303,A -85,B 0,C 180,E1 25051.313,E2 25051.313} C_VEL
LIN {X 0,Y 534.992,Z 290.3,A -85,B 0,C 180,E1 25050.99,E2 25050.99} C_VEL
LIN {X 0,Y 533.49,Z 329.28,A -85,B 0,C 180,E1 25047.697,E2 25047.697} C_VEL
LIN {X 0,Y 533.154,Z 342.603,A -85,B 0,C 180,E1 25046.638,E2 25046.638} C_VEL
LIN {X 0,Y 535.101,Z 355.243,A -85,B 0,C 180,E1 25046.337,E2 25046.337} C_VEL
LIN {X 0,Y 533.574,Z 559.734,A -85,B 0,C 180,E1 25043.414,E2 25043.414} C_VEL
LIN {X 0,Y 533.162,Z 579.368,A -85,B 0,C 180,E1 25042.929,E2 25042.929} C_VEL
LIN {X 0,Y 532.643,Z 598.047,A -85,B 0,C 180,E1 25042.264,E2 25042.264} C_VEL
LIN {X 0,Y 532.045,Z 615.497,A -85,B 0,C 180,E1 25041.439,E2 25041.439} C_VEL
LIN {X 0,Y 531.351,Z 633.357,A -85,B 0,C 180,E1 25040.372,E2 25040.372} C_VEL
LIN {X 0,Y 530.673,Z 650.135,A -85,B 0,C 180,E1 25039.137,E2 25039.137} C_VEL
LIN {X 0,Y 530.001,Z 665.776,A -85,B 0,C 180,E1 25037.732,E2 25037.732} C_VEL
LIN {X 0,Y 529.424,Z 679.736,A -85,B 0,C 180,E1 25036.231,E2 25036.231} C_VEL
LIN {X 0,Y 528.923,Z 692.743,A -85,B 0,C 180,E1 25034.561,E2 25034.561} C_VEL
LIN {X 0,Y 528.529,Z 704.205,A -85,B 0,C 180,E1 25032.787,E2 25032.787} C_VEL
LIN {X 0,Y 528.25,Z 714.139,A -85,B 0,C 180,E1 25030.91,E2 25030.91} C_VEL
LIN {X 0,Y 528.07,Z 722.57,A -85,B 0,C 180,E1 25028.932,E2 25028.932} C_VEL
LIN {X 0,Y 527.969,Z 729.125,A -85,B 0,C 180,E1 25026.961,E2 25026.961} C_VEL
LIN {X 0,Y 527.932,Z 734.152,A -85,B 0,C 180,E1 25024.889,E2 25024.889} C_VEL
LIN {X 0,Y 527.912,Z 737.34,A -85,B 0,C 180,E1 25022.822,E2 25022.822} C_VEL
LIN {X 0,Y 527.917,Z 738.83,A -85,B 0,C 180,E1 25020.759,E2 25020.759} C_VEL
LIN {X 0,Y 527.911,Z 738.671,A -85,B 0,C 180,E1 25018.697,E2 25018.697} C_VEL
LIN {X 0,Y 527.915,Z 736.802,A -85,B 0,C 180,E1 25016.634,E2 25016.634} C_VEL
LIN {X 0,Y 527.932,Z 733.178,A -85,B 0,C 180,E1 25014.566,E2 25014.566} C_VEL
LIN {X 0,Y 527.986,Z 727.754,A -85,B 0,C 180,E1 25012.491,E2 25012.491} C_VEL
LIN {X 0,Y 528.113,Z 720.829,A -85,B 0,C 180,E1 25010.519,E2 25010.519} C_VEL
LIN {X 0,Y 528.317,Z 711.915,A -85,B 0,C 180,E1 25008.538,E2 25008.538} C_VEL
LIN {X 0,Y 528.625,Z 701.393,A -85,B 0,C 180,E1 25006.658,E2 25006.658} C_VEL
LIN {X 0,Y 529.045,Z 689.306,A -85,B 0,C 180,E1 25004.881,E2 25004.881} C_VEL
LIN {X 0,Y 529.58,Z 675.608,A -85,B 0,C 180,E1 25003.209,E2 25003.209} C_VEL
LIN {X 0,Y 530.18,Z 661.357,A -85,B 0,C 180,E1 25001.756,E2 25001.756} C_VEL
LIN {X 0,Y 530.858,Z 645.547,A -85,B 0,C 180,E1 25000.411,E2 25000.411} C_VEL
LIN {X 0,Y 531.552,Z 628.56,A -85,B 0,C 180,E1 24999.227,E2 24999.227} C_VEL
LIN {X 0,Y 532.227,Z 610.564,A -85,B 0,C 180,E1 24998.22,E2 24998.22} C_VEL
LIN {X 0,Y 532.834,Z 591.907,A -85,B 0,C 180,E1 24997.405,E2 24997.405} C_VEL
LIN {X 0,Y 533.31,Z 572.811,A -85,B 0,C 180,E1 24996.794,E2 24996.794} C_VEL
LIN {X 0,Y 533.655,Z 552.956,A -85,B 0,C 180,E1 24996.379,E2 24996.379} C_VEL
LIN {X 0,Y 534.074,Z 493.908,A -85,B 0,C 180,E1 24995.54,E2 24995.54} C_VEL
LIN {X 0,Y 533.205,Z 486.322,A -85,B 0,C 180,E1 24995.388,E2 24995.388} C_VEL
LIN {X 0,Y 527.673,Z 466.49,A -85,B 0,C 180,E1 24994.821,E2 24994.821} C_VEL
LIN {X 0,Y 527.04,Z 459.968,A -85,B 0,C 180,E1 24994.693,E2 24994.693} C_VEL
LIN {X 0,Y 527.743,Z 353.96,A -85,B 0,C 180,E1 24993.156,E2 24993.156} C_VEL
LIN {X 0,Y 525.72,Z 341.772,A -85,B 0,C 180,E1 24992.826,E2 24992.826} C_VEL
LIN {X 0,Y 527.445,Z 297.433,A -85,B 0,C 180,E1 24989.087,E2 24989.087} C_VEL
LIN {X 0,Y 527.649,Z 292.421,A -85,B 0,C 180,E1 24988.657,E2 24988.657} C_VEL
LIN {X 0,Y 520.596,Z 271.913,A -85,B 0,C 180,E1 24986.267,E2 24986.267} C_VEL
LIN {X 0,Y 520.577,Z 271.605,A -85,B 0,C 180,E1 24985.084,E2 24985.084} C_VEL
LIN {X 0,Y 520.553,Z 271.642,A -85,B 0,C 180,E1 24981.654,E2 24981.654} C_VEL
LIN {X 0,Y 520.564,Z 271.635,A -85,B 0,C 180,E1 24978.181,E2 24978.181} C_VEL
LIN {X 0,Y 520.584,Z 271.639,A -85,B 0,C 180,E1 24974.821,E2 24974.821} C_VEL
LIN {X 0,Y 520.589,Z 271.641,A -85,B 0,C 180,E1 24971.325,E2 24971.325} C_VEL
LIN {X 0,Y 520.573,Z 271.64,A -85,B 0,C 180,E1 24967.869,E2 24967.869} C_VEL
LIN {X 0,Y 520.583,Z 271.634,A -85,B 0,C 180,E1 24964.38,E2 24964.38} C_VEL
LIN {X 0,Y 520.561,Z 271.637,A -85,B 0,C 180,E1 24960.982,E2 24960.982} C_VEL
LIN {X 0,Y 520.58,Z 271.642,A -85,B 0,C 180,E1 24957.574,E2 24957.574} C_VEL
LIN {X 0,Y 520.586,Z 271.632,A -85,B 0,C 180,E1 24954.149,E2 24954.149} C_VEL
LIN {X 0,Y 520.544,Z 271.638,A -85,B 0,C 180,E1 24950.816,E2 24950.816} C_VEL
LIN {X 0,Y 520.541,Z 271.645,A -85,B 0,C 180,E1 24947.321,E2 24947.321} C_VEL
LIN {X 0,Y 520.584,Z 271.616,A -85,B 0,C 180,E1 24944.006,E2 24944.006} C_VEL
LIN {X 0,Y 520.528,Z 271.626,A -85,B 0,C 180,E1 24940.627,E2 24940.627} C_VEL
LIN {X 0,Y 520.604,Z 271.906,A -85,B 0,C 180,E1 24939.909,E2 24939.909} C_VEL
LIN {X 0,Y 526.056,Z 289.295,A -85,B 0,C 180,E1 24938.142,E2 24938.142} C_VEL
LIN {X 0,Y 525.617,Z 328.259,A -85,B 0,C 180,E1 24935.021,E2 24935.021} C_VEL
LIN {X 0,Y 524.934,Z 369.946,A -85,B 0,C 180,E1 24931.693,E2 24931.693} C_VEL
LIN {X 0,Y 524.037,Z 413.741,A -85,B 0,C 180,E1 24928.197,E2 24928.197} C_VEL
LIN {X 0,Y 523.081,Z 456.223,A -85,B 0,C 180,E1 24924.804,E2 24924.804} C_VEL
LIN {X 0,Y 522.811,Z 473.835,A -85,B 0,C 180,E1 24923.447,E2 24923.447} C_VEL
LIN {X 0,Y 523.704,Z 483.653,A -85,B 0,C 180,E1 24923.269,E2 24923.269} C_VEL
LIN {X 0,Y 522.921,Z 616.085,A -85,B 0,C 180,E1 24921.396,E2 24921.396} C_VEL
LIN {X 0,Y 522.693,Z 631.969,A -85,B 0,C 180,E1 24920.973,E2 24920.973} C_VEL
LIN {X 0,Y 522.333,Z 648.53,A -85,B 0,C 180,E1 24920.304,E2 24920.304} C_VEL
LIN {X 0,Y 521.931,Z 662.754,A -85,B 0,C 180,E1 24919.516,E2 24919.516} C_VEL
LIN {X 0,Y 521.46,Z 677.361,A -85,B 0,C 180,E1 24918.468,E2 24918.468} C_VEL
LIN {X 0,Y 521.044,Z 690.15,A -85,B 0,C 180,E1 24917.299,E2 24917.299} C_VEL
LIN {X 0,Y 520.675,Z 701.58,A -85,B 0,C 180,E1 24915.999,E2 24915.999} C_VEL
LIN {X 0,Y 520.383,Z 711.333,A -85,B 0,C 180,E1 24914.625,E2 24914.625} C_VEL
LIN {X 0,Y 520.152,Z 720.372,A -85,B 0,C 180,E1 24913.013,E2 24913.013} C_VEL
LIN {X 0,Y 520.018,Z 727.428,A -85,B 0,C 180,E1 24911.389,E2 24911.389} C_VEL
LIN {X 0,Y 519.946,Z 732.976,A -85,B 0,C 180,E1 24909.633,E2 24909.633} C_VEL
LIN {X 0,Y 519.924,Z 736.732,A -85,B 0,C 180,E1 24907.858,E2 24907.858} C_VEL
LIN {X 0,Y 519.917,Z 738.705,A -85,B 0,C 180,E1 24905.992,E2 24905.992} C_VEL
LIN {X 0,Y 519.916,Z 738.85,A -85,B 0,C 180,E1 24904.162,E2 24904.162} C_VEL
LIN {X 0,Y 519.919,Z 737.028,A -85,B 0,C 180,E1 24902.266,E2 24902.266} C_VEL
LIN {X 0,Y 519.941,Z 733.601,A -85,B 0,C 180,E1 24900.51,E2 24900.51} C_VEL
LIN {X 0,Y 520.007,Z 728.163,A -85,B 0,C 180,E1 24898.727,E2 24898.727} C_VEL
LIN {X 0,Y 520.139,Z 721.127,A -85,B 0,C 180,E1 24897.045,E2 24897.045} C_VEL
LIN {X 0,Y 520.364,Z 712.036,A -85,B 0,C 180,E1 24895.397,E2 24895.397} C_VEL
LIN {X 0,Y 520.667,Z 701.897,A -85,B 0,C 180,E1 24893.947,E2 24893.947} C_VEL
LIN {X 0,Y 521.073,Z 689.476,A -85,B 0,C 180,E1 24892.537,E2 24892.537} C_VEL
LIN {X 0,Y 521.491,Z 676.573,A -85,B 0,C 180,E1 24891.377,E2 24891.377} C_VEL
LIN {X 0,Y 521.942,Z 662.32,A -85,B 0,C 180,E1 24890.363,E2 24890.363} C_VEL
LIN {X 0,Y 522.345,Z 648.167,A -85,B 0,C 180,E1 24889.588,E2 24889.588} C_VEL
LIN {X 0,Y 522.701,Z 631.66,A -85,B 0,C 180,E1 24888.924,E2 24888.924} C_VEL
LIN {X 0,Y 522.914,Z 615.706,A -85,B 0,C 180,E1 24888.505,E2 24888.505} C_VEL
LIN {X 0,Y 523.514,Z 479.738,A -85,B 0,C 180,E1 24886.578,E2 24886.578} C_VEL
LIN {X 0,Y 522.734,Z 473.073,A -85,B 0,C 180,E1 24886.424,E2 24886.424} C_VEL
LIN {X 0,Y 523.654,Z 429.594,A -85,B 0,C 180,E1 24882.974,E2 24882.974} C_VEL
LIN {X 0,Y 524.395,Z 391.914,A -85,B 0,C 180,E1 24879.983,E2 24879.983} C_VEL
LIN {X 0,Y 525.069,Z 354.99,A -85,B 0,C 180,E1 24877.075,E2 24877.075} C_VEL
LIN {X 0,Y 525.468,Z 315.98,A -85,B 0,C 180,E1 24874.016,E2 24874.016} C_VEL
LIN {X 0,Y 525.494,Z 287.797,A -85,B 0,C 180,E1 24871.807,E2 24871.807} C_VEL
LIN {X 0,Y 520.607,Z 272.052,A -85,B 0,C 180,E1 24870.275,E2 24870.275} C_VEL
LIN {X 0,Y 520.567,Z 271.642,A -85,B 0,C 180,E1 24869.96,E2 24869.96} C_VEL
LIN {X 0,Y 520.543,Z 271.643,A -85,B 0,C 180,E1 24866.587,E2 24866.587} C_VEL
LIN {X 0,Y 520.579,Z 271.64,A -85,B 0,C 180,E1 24863.188,E2 24863.188} C_VEL
LIN {X 0,Y 520.578,Z 271.644,A -85,B 0,C 180,E1 24859.758,E2 24859.758} C_VEL
LIN {X 0,Y 520.542,Z 271.642,A -85,B 0,C 180,E1 24856.401,E2 24856.401} C_VEL
LIN {X 0,Y 520.57,Z 271.638,A -85,B 0,C 180,E1 24852.987,E2 24852.987} C_VEL
LIN {X 0,Y 520.587,Z 271.641,A -85,B 0,C 180,E1 24849.508,E2 24849.508} C_VEL
LIN {X 0,Y 520.546,Z 271.64,A -85,B 0,C 180,E1 24846.175,E2 24846.175} C_VEL
LIN {X 0,Y 520.561,Z 271.638,A -85,B 0,C 180,E1 24842.753,E2 24842.753} C_VEL
LIN {X 0,Y 520.59,Z 271.638,A -85,B 0,C 180,E1 24839.34,E2 24839.34} C_VEL
LIN {X 0,Y 520.554,Z 271.64,A -85,B 0,C 180,E1 24835.925,E2 24835.925} C_VEL
LIN {X 0,Y 520.552,Z 271.638,A -85,B 0,C 180,E1 24832.384,E2 24832.384} C_VEL
LIN {X 0,Y 520.587,Z 271.637,A -85,B 0,C 180,E1 24829.039,E2 24829.039} C_VEL
LIN {X 0,Y 520.574,Z 271.642,A -85,B 0,C 180,E1 24825.541,E2 24825.541} C_VEL
LIN {X 0,Y 520.549,Z 271.639,A -85,B 0,C 180,E1 24822.102,E2 24822.102} C_VEL
LIN {X 0,Y 520.578,Z 271.634,A -85,B 0,C 180,E1 24818.669,E2 24818.669} C_VEL
LIN {X 0,Y 520.587,Z 271.64,A -85,B 0,C 180,E1 24815.248,E2 24815.248} C_VEL
LIN {X 0,Y 520.554,Z 271.64,A -85,B 0,C 180,E1 24811.803,E2 24811.803} C_VEL
LIN {X 0,Y 520.558,Z 271.637,A -85,B 0,C 180,E1 24808.246,E2 24808.246} C_VEL
LIN {X 0,Y 520.587,Z 271.637,A -85,B 0,C 180,E1 24804.817,E2 24804.817} C_VEL
LIN {X 0,Y 520.573,Z 271.642,A -85,B 0,C 180,E1 24801.375,E2 24801.375} C_VEL
LIN {X 0,Y 520.554,Z 271.64,A -85,B 0,C 180,E1 24797.907,E2 24797.907} C_VEL
LIN {X 0,Y 520.584,Z 271.637,A -85,B 0,C 180,E1 24794.508,E2 24794.508} C_VEL
LIN {X 0,Y 520.589,Z 271.641,A -85,B 0,C 180,E1 24790.992,E2 24790.992} C_VEL
LIN {X 0,Y 520.553,Z 271.631,A -85,B 0,C 180,E1 24787.645,E2 24787.645} C_VEL
LIN {X 0,Y 520.609,Z 271.883,A -85,B 0,C 180,E1 24786.232,E2 24786.232} C_VEL
LIN {X 0,Y 522.835,Z 277.781,A -85,B 0,C 180,E1 24785.544,E2 24785.544} C_VEL
LIN {X 0,Y 529.438,Z 295.079,A -85,B 0,C 180,E1 24783.724,E2 24783.724} C_VEL
LIN {X 0,Y 528.74,Z 316.137,A -85,B 0,C 180,E1 24782.208,E2 24782.208} C_VEL
LIN {X 0,Y 530.995,Z 330.738,A -85,B 0,C 180,E1 24781.837,E2 24781.837} C_VEL
LIN {X 0,Y 529.192,Z 533.372,A -85,B 0,C 180,E1 24778.875,E2 24778.875} C_VEL
LIN {X 0,Y 528.748,Z 578.449,A -85,B 0,C 180,E1 24778.196,E2 24778.196} C_VEL
LIN {X 0,Y 528.168,Z 599.563,A -85,B 0,C 180,E1 24777.669,E2 24777.669} C_VEL
LIN {X 0,Y 527.46,Z 619.053,A -85,B 0,C 180,E1 24776.979,E2 24776.979} C_VEL
LIN {X 0,Y 526.617,Z 638.315,A -85,B 0,C 180,E1 24776.096,E2 24776.096} C_VEL
LIN {X 0,Y 525.65,Z 657.848,A -85,B 0,C 180,E1 24774.977,E2 24774.977} C_VEL
LIN {X 0,Y 524.688,Z 675.99,A -85,B 0,C 180,E1 24773.707,E2 24773.707} C_VEL
LIN {X 0,Y 523.735,Z 693.189,A -85,B 0,C 180,E1 24772.267,E2 24772.267} C_VEL
LIN {X 0,Y 522.831,Z 709.385,A -85,B 0,C 180,E1 24770.659,E2 24770.659} C_VEL
LIN {X 0,Y 522.006,Z 724.518,A -85,B 0,C 180,E1 24768.878,E2 24768.878} C_VEL
LIN {X 0,Y 521.321,Z 738.359,A -85,B 0,C 180,E1 24766.948,E2 24766.948} C_VEL
LIN {X 0,Y 520.808,Z 750.021,A -85,B 0,C 180,E1 24765.02,E2 24765.02} C_VEL
LIN {X 0,Y 520.406,Z 760.854,A -85,B 0,C 180,E1 24762.876,E2 24762.876} C_VEL
LIN {X 0,Y 520.153,Z 770.066,A -85,B 0,C 180,E1 24760.633,E2 24760.633} C_VEL
LIN {X 0,Y 520.012,Z 777.295,A -85,B 0,C 180,E1 24758.401,E2 24758.401} C_VEL
LIN {X 0,Y 519.946,Z 782.733,A -85,B 0,C 180,E1 24756.179,E2 24756.179} C_VEL
LIN {X 0,Y 519.919,Z 786.405,A -85,B 0,C 180,E1 24753.969,E2 24753.969} C_VEL
LIN {X 0,Y 519.907,Z 788.443,A -85,B 0,C 180,E1 24751.762,E2 24751.762} C_VEL
LIN {X 0,Y 519.9,Z 788.895,A -85,B 0,C 180,E1 24749.448,E2 24749.448} C_VEL
LIN {X 0,Y 519.911,Z 787.729,A -85,B 0,C 180,E1 24747.243,E2 24747.243} C_VEL
LIN {X 0,Y 519.92,Z 784.881,A -85,B 0,C 180,E1 24744.979,E2 24744.979} C_VEL
LIN {X 0,Y 519.953,Z 780.479,A -85,B 0,C 180,E1 24742.818,E2 24742.818} C_VEL
LIN {X 0,Y 520.044,Z 774.616,A -85,B 0,C 180,E1 24740.705,E2 24740.705} C_VEL
LIN {X 0,Y 520.225,Z 767.086,A -85,B 0,C 180,E1 24738.58,E2 24738.58} C_VEL
LIN {X 0,Y 520.523,Z 757.703,A -85,B 0,C 180,E1 24736.446,E2 24736.446} C_VEL
LIN {X 0,Y 520.943,Z 746.823,A -85,B 0,C 180,E1 24734.412,E2 24734.412} C_VEL
LIN {X 0,Y 521.506,Z 734.493,A -85,B 0,C 180,E1 24732.481,E2 24732.481} C_VEL
LIN {X 0,Y 522.2,Z 720.731,A -85,B 0,C 180,E1 24730.655,E2 24730.655} C_VEL
LIN {X 0,Y 523.025,Z 705.489,A -85,B 0,C 180,E1 24728.936,E2 24728.936} C_VEL
LIN {X 0,Y 523.971,Z 688.603,A -85,B 0,C 180,E1 24727.327,E2 24727.327} C_VEL
LIN {X 0,Y 524.948,Z 671.36,A -85,B 0,C 180,E1 24725.945,E2 24725.945} C_VEL
LIN {X 0,Y 525.91,Z 653.42,A -85,B 0,C 180,E1 24724.743,E2 24724.743} C_VEL
LIN {X 0,Y 526.807,Z 634.182,A -85,B 0,C 180,E1 24723.693,E2 24723.693} C_VEL
LIN {X 0,Y 527.624,Z 614.8,A -85,B 0,C 180,E1 24722.855,E2 24722.855} C_VEL
LIN {X 0,Y 528.309,Z 594.391,A -85,B 0,C 180,E1 24722.187,E2 24722.187} C_VEL
LIN {X 0,Y 528.817,Z 573.178,A -85,B 0,C 180,E1 24721.71,E2 24721.71} C_VEL
LIN {X 0,Y 530.518,Z 341.093,A -85,B 0,C 180,E1 24718.394,E2 24718.394} C_VEL
LIN {X 0,Y 530.379,Z 327.998,A -85,B 0,C 180,E1 24718.19,E2 24718.19} C_VEL
LIN {X 0,Y 528.39,Z 316.056,A -85,B 0,C 180,E1 24717.877,E2 24717.877} C_VEL
LIN {X 0,Y 528.883,Z 294.028,A -85,B 0,C 180,E1 24716.286,E2 24716.286} C_VEL
LIN {X 0,Y 521.663,Z 274.863,A -85,B 0,C 180,E1 24714.263,E2 24714.263} C_VEL
LIN {X 0,Y 520.597,Z 271.853,A -85,B 0,C 180,E1 24713.869,E2 24713.869} C_VEL
LIN {X 0,Y 520.551,Z 271.644,A -85,B 0,C 180,E1 24710.374,E2 24710.374} C_VEL
LIN {X 0,Y 520.584,Z 271.642,A -85,B 0,C 180,E1 24707.012,E2 24707.012} C_VEL
LIN {X 0,Y 520.575,Z 271.641,A -85,B 0,C 180,E1 24703.592,E2 24703.592} C_VEL
LIN {X 0,Y 520.543,Z 271.645,A -85,B 0,C 180,E1 24700.194,E2 24700.194} C_VEL
LIN {X 0,Y 520.569,Z 271.644,A -85,B 0,C 180,E1 24696.78,E2 24696.78} C_VEL
LIN {X 0,Y 520.577,Z 271.875,A -85,B 0,C 180,E1 24693.898,E2 24693.898} C_VEL
LIN {X 0,Y 524.315,Z 282.062,A -85,B 0,C 180,E1 24692.553,E2 24692.553} C_VEL
LIN {X 0,Y 527.874,Z 293.038,A -85,B 0,C 180,E1 24691.264,E2 24691.264} C_VEL
LIN {X 0,Y 525.988,Z 334.41,A -85,B 0,C 180,E1 24687.695,E2 24687.695} C_VEL
LIN {X 0,Y 525.771,Z 342.541,A -85,B 0,C 180,E1 24687.045,E2 24687.045} C_VEL
LIN {X 0,Y 527.928,Z 356.398,A -85,B 0,C 180,E1 24686.707,E2 24686.707} C_VEL
LIN {X 0,Y 526.234,Z 559.761,A -85,B 0,C 180,E1 24683.761,E2 24683.761} C_VEL
LIN {X 0,Y 525.776,Z 579.393,A -85,B 0,C 180,E1 24683.27,E2 24683.27} C_VEL
LIN {X 0,Y 525.193,Z 598.474,A -85,B 0,C 180,E1 24682.579,E2 24682.579} C_VEL
LIN {X 0,Y 524.498,Z 616.529,A -85,B 0,C 180,E1 24681.704,E2 24681.704} C_VEL
LIN {X 0,Y 523.739,Z 634.212,A -85,B 0,C 180,E1 24680.623,E2 24680.623} C_VEL
LIN {X 0,Y 523.02,Z 650.143,A -85,B 0,C 180,E1 24679.429,E2 24679.429} C_VEL
LIN {X 0,Y 522.275,Z 665.726,A -85,B 0,C 180,E1 24678.01,E2 24678.01} C_VEL
LIN {X 0,Y 521.623,Z 679.741,A -85,B 0,C 180,E1 24676.48,E2 24676.48} C_VEL
LIN {X 0,Y 521.059,Z 692.752,A -85,B 0,C 180,E1 24674.786,E2 24674.786} C_VEL
LIN {X 0,Y 520.616,Z 704.206,A -85,B 0,C 180,E1 24672.985,E2 24672.985} C_VEL
LIN {X 0,Y 520.299,Z 714.139,A -85,B 0,C 180,E1 24671.079,E2 24671.079} C_VEL
LIN {X 0,Y 520.094,Z 722.571,A -85,B 0,C 180,E1 24669.07,E2 24669.07} C_VEL
LIN {X 0,Y 519.98,Z 729.129,A -85,B 0,C 180,E1 24667.069,E2 24667.069} C_VEL
LIN {X 0,Y 519.934,Z 734.156,A -85,B 0,C 180,E1 24664.964,E2 24664.964} C_VEL
LIN {X 0,Y 519.913,Z 737.337,A -85,B 0,C 180,E1 24662.866,E2 24662.866} C_VEL
LIN {X 0,Y 519.917,Z 738.829,A -85,B 0,C 180,E1 24660.771,E2 24660.771} C_VEL
LIN {X 0,Y 519.911,Z 738.672,A -85,B 0,C 180,E1 24658.677,E2 24658.677} C_VEL
LIN {X 0,Y 519.914,Z 736.798,A -85,B 0,C 180,E1 24656.582,E2 24656.582} C_VEL
LIN {X 0,Y 519.936,Z 733.173,A -85,B 0,C 180,E1 24654.482,E2 24654.482} C_VEL
LIN {X 0,Y 519.996,Z 727.749,A -85,B 0,C 180,E1 24652.375,E2 24652.375} C_VEL
LIN {X 0,Y 520.14,Z 720.827,A -85,B 0,C 180,E1 24650.372,E2 24650.372} C_VEL
LIN {X 0,Y 520.373,Z 711.91,A -85,B 0,C 180,E1 24648.36,E2 24648.36} C_VEL
LIN {X 0,Y 520.72,Z 701.384,A -85,B 0,C 180,E1 24646.452,E2 24646.452} C_VEL
LIN {X 0,Y 521.195,Z 689.297,A -85,B 0,C 180,E1 24644.648,E2 24644.648} C_VEL
LIN {X 0,Y 521.799,Z 675.599,A -85,B 0,C 180,E1 24642.951,E2 24642.951} C_VEL
LIN {X 0,Y 522.47,Z 661.351,A -85,B 0,C 180,E1 24641.477,E2 24641.477} C_VEL
LIN {X 0,Y 523.246,Z 645.093,A -85,B 0,C 180,E1 24640.078,E2 24640.078} C_VEL
LIN {X 0,Y 523.989,Z 628.721,A -85,B 0,C 180,E1 24638.923,E2 24638.923} C_VEL
LIN {X 0,Y 524.744,Z 610.55,A -85,B 0,C 180,E1 24637.894,E2 24637.894} C_VEL
LIN {X 0,Y 525.405,Z 592.299,A -85,B 0,C 180,E1 24637.083,E2 24637.083} C_VEL
LIN {X 0,Y 525.935,Z 573.232,A -85,B 0,C 180,E1 24636.461,E2 24636.461} C_VEL
LIN {X 0,Y 526.317,Z 553.452,A -85,B 0,C 180,E1 24636.039,E2 24636.039} C_VEL
LIN {X 0,Y 527.04,Z 459.968,A -85,B 0,C 180,E1 24634.693,E2 24634.693} C_VEL
LIN {X 0,Y 526.195,Z 452.38,A -85,B 0,C 180,E1 24634.537,E2 24634.537} C_VEL
LIN {X 0,Y 520.736,Z 432.549,A -85,B 0,C 180,E1 24633.954,E2 24633.954} C_VEL
LIN {X 0,Y 520.123,Z 426.027,A -85,B 0,C 180,E1 24633.823,E2 24633.823} C_VEL
LIN {X 0,Y 520.602,Z 355.073,A -85,B 0,C 180,E1 24632.77,E2 24632.77} C_VEL
LIN {X 0,Y 518.426,Z 341.796,A -85,B 0,C 180,E1 24632.396,E2 24632.396} C_VEL
LIN {X 0,Y 520.253,Z 299.007,A -85,B 0,C 180,E1 24628.741,E2 24628.741} C_VEL
LIN {X 0,Y 520.238,Z 294.715,A -85,B 0,C 180,E1 24628.352,E2 24628.352} C_VEL
LIN {X 0,Y 513.404,Z 275.245,A -85,B 0,C 180,E1 24626.063,E2 24626.063} C_VEL
LIN {X 0,Y 512.629,Z 272.811,A -85,B 0,C 180,E1 24625.723,E2 24625.723} C_VEL
LIN {X 0,Y 512.641,Z 272.625,A -85,B 0,C 180,E1 24622.516,E2 24622.516} C_VEL
LIN {X 0,Y 512.649,Z 272.627,A -85,B 0,C 180,E1 24619.009,E2 24619.009} C_VEL
LIN {X 0,Y 512.631,Z 272.627,A -85,B 0,C 180,E1 24615.551,E2 24615.551} C_VEL
LIN {X 0,Y 512.63,Z 272.628,A -85,B 0,C 180,E1 24611.991,E2 24611.991} C_VEL
LIN {X 0,Y 512.649,Z 272.624,A -85,B 0,C 180,E1 24608.476,E2 24608.476} C_VEL
LIN {X 0,Y 512.631,Z 272.628,A -85,B 0,C 180,E1 24604.991,E2 24604.991} C_VEL
LIN {X 0,Y 512.644,Z 272.63,A -85,B 0,C 180,E1 24601.515,E2 24601.515} C_VEL
LIN {X 0,Y 512.648,Z 272.623,A -85,B 0,C 180,E1 24598.038,E2 24598.038} C_VEL
LIN {X 0,Y 512.627,Z 272.62,A -85,B 0,C 180,E1 24594.549,E2 24594.549} C_VEL
LIN {X 0,Y 512.605,Z 272.627,A -85,B 0,C 180,E1 24591.153,E2 24591.153} C_VEL
LIN {X 0,Y 512.64,Z 272.625,A -85,B 0,C 180,E1 24587.832,E2 24587.832} C_VEL
LIN {X 0,Y 512.61,Z 272.609,A -85,B 0,C 180,E1 24584.459,E2 24584.459} C_VEL
LIN {X 0,Y 512.577,Z 272.624,A -85,B 0,C 180,E1 24581.131,E2 24581.131} C_VEL
LIN {X 0,Y 512.662,Z 272.926,A -85,B 0,C 180,E1 24580.309,E2 24580.309} C_VEL
LIN {X 0,Y 518.697,Z 292.075,A -85,B 0,C 180,E1 24578.342,E2 24578.342} C_VEL
LIN {X 0,Y 518.15,Z 331.621,A -85,B 0,C 180,E1 24575.149,E2 24575.149} C_VEL
LIN {X 0,Y 517.386,Z 372.895,A -85,B 0,C 180,E1 24571.828,E2 24571.828} C_VEL
LIN {X 0,Y 516.402,Z 417.038,A -85,B 0,C 180,E1 24568.281,E2 24568.281} C_VEL
LIN {X 0,Y 515.379,Z 461.419,A -85,B 0,C 180,E1 24564.714,E2 24564.714} C_VEL
LIN {X 0,Y 515.161,Z 474.189,A -85,B 0,C 180,E1 24563.727,E2 24563.727} C_VEL
LIN {X 0,Y 516.114,Z 484.411,A -85,B 0,C 180,E1 24563.539,E2 24563.539} C_VEL
LIN {X 0,Y 515.251,Z 616.503,A -85,B 0,C 180,E1 24561.643,E2 24561.643} C_VEL
LIN {X 0,Y 515.005,Z 632.345,A -85,B 0,C 180,E1 24561.215,E2 24561.215} C_VEL
LIN {X 0,Y 514.623,Z 648.552,A -85,B 0,C 180,E1 24560.552,E2 24560.552} C_VEL
LIN {X 0,Y 514.176,Z 663.264,A -85,B 0,C 180,E1 24559.728,E2 24559.728} C_VEL
LIN {X 0,Y 513.662,Z 677.86,A -85,B 0,C 180,E1 24558.663,E2 24558.663} C_VEL
LIN {X 0,Y 513.218,Z 690.291,A -85,B 0,C 180,E1 24557.512,E2 24557.512} C_VEL
LIN {X 0,Y 512.785,Z 702.303,A -85,B 0,C 180,E1 24556.125,E2 24556.125} C_VEL
LIN {X 0,Y 512.461,Z 711.979,A -85,B 0,C 180,E1 24554.73,E2 24554.73} C_VEL
LIN {X 0,Y 512.198,Z 721.204,A -85,B 0,C 180,E1 24553.046,E2 24553.046} C_VEL
LIN {X 0,Y 512.048,Z 727.969,A -85,B 0,C 180,E1 24551.442,E2 24551.442} C_VEL
LIN {X 0,Y 511.963,Z 733.565,A -85,B 0,C 180,E1 24549.627,E2 24549.627} C_VEL
LIN {X 0,Y 511.936,Z 737.182,A -85,B 0,C 180,E1 24547.857,E2 24547.857} C_VEL
LIN {X 0,Y 511.927,Z 739.08,A -85,B 0,C 180,E1 24546.032,E2 24546.032} C_VEL
LIN {X 0,Y 511.926,Z 739.258,A -85,B 0,C 180,E1 24544.182,E2 24544.182} C_VEL
LIN {X 0,Y 511.931,Z 737.529,A -85,B 0,C 180,E1 24542.302,E2 24542.302} C_VEL
LIN {X 0,Y 511.959,Z 734.186,A -85,B 0,C 180,E1 24540.519,E2 24540.519} C_VEL
LIN {X 0,Y 512.028,Z 729.131,A -85,B 0,C 180,E1 24538.794,E2 24538.794} C_VEL
LIN {X 0,Y 512.176,Z 722.266,A -85,B 0,C 180,E1 24537.082,E2 24537.082} C_VEL
LIN {X 0,Y 512.399,Z 714.171,A -85,B 0,C 180,E1 24535.538,E2 24535.538} C_VEL
LIN {X 0,Y 512.724,Z 704.172,A -85,B 0,C 180,E1 24534.027,E2 24534.027} C_VEL
LIN {X 0,Y 513.121,Z 693.219,A -85,B 0,C 180,E1 24532.701,E2 24532.701} C_VEL
LIN {X 0,Y 513.602,Z 679.796,A -85,B 0,C 180,E1 24531.405,E2 24531.405} C_VEL
LIN {X 0,Y 514.085,Z 666.102,A -85,B 0,C 180,E1 24530.364,E2 24530.364} C_VEL
LIN {X 0,Y 514.554,Z 651.211,A -85,B 0,C 180,E1 24529.487,E2 24529.487} C_VEL
LIN {X 0,Y 514.943,Z 635.865,A -85,B 0,C 180,E1 24528.817,E2 24528.817} C_VEL
LIN {X 0,Y 515.215,Z 619.068,A -85,B 0,C 180,E1 24528.32,E2 24528.32} C_VEL
LIN {X 0,Y 515.387,Z 595.185,A -85,B 0,C 180,E1 24527.936,E2 24527.936} C_VEL
LIN {X 0,Y 515.916,Z 480.468,A -85,B 0,C 180,E1 24526.305,E2 24526.305} C_VEL
LIN {X 0,Y 515.086,Z 473.319,A -85,B 0,C 180,E1 24526.135,E2 24526.135} C_VEL
LIN {X 0,Y 516.078,Z 429.056,A -85,B 0,C 180,E1 24522.592,E2 24522.592} C_VEL
LIN {X 0,Y 516.988,Z 388.843,A -85,B 0,C 180,E1 24519.373,E2 24519.373} C_VEL
LIN {X 0,Y 517.686,Z 347.255,A -85,B 0,C 180,E1 24516.092,E2 24516.092} C_VEL
LIN {X 0,Y 518.126,Z 307.146,A -85,B 0,C 180,E1 24512.922,E2 24512.922} C_VEL
LIN {X 0,Y 518.1,Z 290.356,A -85,B 0,C 180,E1 24511.599,E2 24511.599} C_VEL
LIN {X 0,Y 512.693,Z 273.013,A -85,B 0,C 180,E1 24509.887,E2 24509.887} C_VEL
LIN {X 0,Y 512.654,Z 272.631,A -85,B 0,C 180,E1 24509.562,E2 24509.562} C_VEL
LIN {X 0,Y 512.614,Z 272.635,A -85,B 0,C 180,E1 24506.156,E2 24506.156} C_VEL
LIN {X 0,Y 512.607,Z 272.631,A -85,B 0,C 180,E1 24502.695,E2 24502.695} C_VEL
LIN {X 0,Y 512.645,Z 272.624,A -85,B 0,C 180,E1 24499.246,E2 24499.246} C_VEL
LIN {X 0,Y 512.639,Z 272.627,A -85,B 0,C 180,E1 24495.731,E2 24495.731} C_VEL
LIN {X 0,Y 512.606,Z 272.63,A -85,B 0,C 180,E1 24492.276,E2 24492.276} C_VEL
LIN {X 0,Y 512.619,Z 272.626,A -85,B 0,C 180,E1 24488.751,E2 24488.751} C_VEL
LIN {X 0,Y 512.649,Z 272.629,A -85,B 0,C 180,E1 24485.372,E2 24485.372} C_VEL
LIN {X 0,Y 512.618,Z 272.631,A -85,B 0,C 180,E1 24481.901,E2 24481.901} C_VEL
LIN {X 0,Y 512.61,Z 272.626,A -85,B 0,C 180,E1 24478.436,E2 24478.436} C_VEL
LIN {X 0,Y 512.644,Z 272.626,A -85,B 0,C 180,E1 24474.965,E2 24474.965} C_VEL
LIN {X 0,Y 512.646,Z 272.63,A -85,B 0,C 180,E1 24471.421,E2 24471.421} C_VEL
LIN {X 0,Y 512.613,Z 272.629,A -85,B 0,C 180,E1 24467.954,E2 24467.954} C_VEL
LIN {X 0,Y 512.615,Z 272.625,A -85,B 0,C 180,E1 24464.385,E2 24464.385} C_VEL
LIN {X 0,Y 512.649,Z 272.626,A -85,B 0,C 180,E1 24460.992,E2 24460.992} C_VEL
LIN {X 0,Y 512.633,Z 272.629,A -85,B 0,C 180,E1 24457.525,E2 24457.525} C_VEL
LIN {X 0,Y 512.612,Z 272.628,A -85,B 0,C 180,E1 24454.047,E2 24454.047} C_VEL
LIN {X 0,Y 512.639,Z 272.623,A -85,B 0,C 180,E1 24450.561,E2 24450.561} C_VEL
LIN {X 0,Y 512.649,Z 272.629,A -85,B 0,C 180,E1 24447.033,E2 24447.033} C_VEL
LIN {X 0,Y 512.619,Z 272.63,A -85,B 0,C 180,E1 24443.634,E2 24443.634} C_VEL
LIN {X 0,Y 512.619,Z 272.627,A -85,B 0,C 180,E1 24440.081,E2 24440.081} C_VEL
LIN {X 0,Y 512.648,Z 272.628,A -85,B 0,C 180,E1 24436.644,E2 24436.644} C_VEL
LIN {X 0,Y 512.643,Z 272.631,A -85,B 0,C 180,E1 24433.16,E2 24433.16} C_VEL
LIN {X 0,Y 512.615,Z 272.631,A -85,B 0,C 180,E1 24429.772,E2 24429.772} C_VEL
LIN {X 0,Y 512.681,Z 272.863,A -85,B 0,C 180,E1 24426.783,E2 24426.783} C_VEL
LIN {X 0,Y 514.781,Z 278.552,A -85,B 0,C 180,E1 24426.1,E2 24426.1} C_VEL
LIN {X 0,Y 522.312,Z 298.215,A -85,B 0,C 180,E1 24423.983,E2 24423.983} C_VEL
LIN {X 0,Y 521.644,Z 316.225,A -85,B 0,C 180,E1 24422.669,E2 24422.669} C_VEL
LIN {X 0,Y 524.062,Z 331.98,A -85,B 0,C 180,E1 24422.257,E2 24422.257} C_VEL
LIN {X 0,Y 522.004,Z 524.959,A -85,B 0,C 180,E1 24419.365,E2 24419.365} C_VEL
LIN {X 0,Y 521.467,Z 578.492,A -85,B 0,C 180,E1 24418.56,E2 24418.56} C_VEL
LIN {X 0,Y 520.875,Z 600.034,A -85,B 0,C 180,E1 24418.026,E2 24418.026} C_VEL
LIN {X 0,Y 520.123,Z 620.862,A -85,B 0,C 180,E1 24417.287,E2 24417.287} C_VEL
LIN {X 0,Y 519.281,Z 639.847,A -85,B 0,C 180,E1 24416.408,E2 24416.408} C_VEL
LIN {X 0,Y 518.247,Z 658.777,A -85,B 0,C 180,E1 24415.295,E2 24415.295} C_VEL
LIN {X 0,Y 517.144,Z 677.456,A -85,B 0,C 180,E1 24413.953,E2 24413.953} C_VEL
LIN {X 0,Y 516.143,Z 693.796,A -85,B 0,C 180,E1 24412.553,E2 24412.553} C_VEL
LIN {X 0,Y 515.145,Z 709.904,A -85,B 0,C 180,E1 24410.922,E2 24410.922} C_VEL
LIN {X 0,Y 514.219,Z 725.369,A -85,B 0,C 180,E1 24409.065,E2 24409.065} C_VEL
LIN {X 0,Y 513.443,Z 739.579,A -85,B 0,C 180,E1 24407.03,E2 24407.03} C_VEL
LIN {X 0,Y 512.849,Z 751.925,A -85,B 0,C 180,E1 24404.911,E2 24404.911} C_VEL
LIN {X 0,Y 512.439,Z 761.882,A -85,B 0,C 180,E1 24402.851,E2 24402.851} C_VEL
LIN {X 0,Y 512.173,Z 770.471,A -85,B 0,C 180,E1 24400.686,E2 24400.686} C_VEL
LIN {X 0,Y 512.019,Z 777.598,A -85,B 0,C 180,E1 24398.42,E2 24398.42} C_VEL
LIN {X 0,Y 511.948,Z 782.936,A -85,B 0,C 180,E1 24396.165,E2 24396.165} C_VEL
LIN {X 0,Y 511.918,Z 786.563,A -85,B 0,C 180,E1 24393.919,E2 24393.919} C_VEL
LIN {X 0,Y 511.904,Z 788.51,A -85,B 0,C 180,E1 24391.678,E2 24391.678} C_VEL
LIN {X 0,Y 511.9,Z 788.895,A -85,B 0,C 180,E1 24389.439,E2 24389.439} C_VEL
LIN {X 0,Y 511.911,Z 787.73,A -85,B 0,C 180,E1 24387.2,E2 24387.2} C_VEL
LIN {X 0,Y 511.92,Z 784.945,A -85,B 0,C 180,E1 24384.942,E2 24384.942} C_VEL
LIN {X 0,Y 511.96,Z 780.479,A -85,B 0,C 180,E1 24382.706,E2 24382.706} C_VEL
LIN {X 0,Y 512.078,Z 774.263,A -85,B 0,C 180,E1 24380.445,E2 24380.445} C_VEL
LIN {X 0,Y 512.293,Z 766.172,A -85,B 0,C 180,E1 24378.173,E2 24378.173} C_VEL
LIN {X 0,Y 512.637,Z 756.556,A -85,B 0,C 180,E1 24376.003,E2 24376.003} C_VEL
LIN {X 0,Y 513.141,Z 745.479,A -85,B 0,C 180,E1 24373.936,E2 24373.936} C_VEL
LIN {X 0,Y 513.792,Z 732.943,A -85,B 0,C 180,E1 24371.975,E2 24371.975} C_VEL
LIN {X 0,Y 514.601,Z 718.86,A -85,B 0,C 180,E1 24370.119,E2 24370.119} C_VEL
LIN {X 0,Y 515.516,Z 703.77,A -85,B 0,C 180,E1 24368.429,E2 24368.429} C_VEL
LIN {X 0,Y 516.554,Z 687.043,A -85,B 0,C 180,E1 24366.842,E2 24366.842} C_VEL
LIN {X 0,Y 517.654,Z 668.921,A -85,B 0,C 180,E1 24365.401,E2 24365.401} C_VEL
LIN {X 0,Y 518.736,Z 650.255,A -85,B 0,C 180,E1 24364.175,E2 24364.175} C_VEL
LIN {X 0,Y 519.635,Z 632.605,A -85,B 0,C 180,E1 24363.228,E2 24363.228} C_VEL
LIN {X 0,Y 520.342,Z 613.516,A -85,B 0,C 180,E1 24362.443,E2 24362.443} C_VEL
LIN {X 0,Y 520.963,Z 593.158,A -85,B 0,C 180,E1 24361.814,E2 24361.814} C_VEL
LIN {X 0,Y 521.396,Z 571.634,A -85,B 0,C 180,E1 24361.36,E2 24361.36} C_VEL
LIN {X 0,Y 522.992,Z 374.414,A -85,B 0,C 180,E1 24358.516,E2 24358.516} C_VEL
LIN {X 0,Y 523.224,Z 329.363,A -85,B 0,C 180,E1 24357.824,E2 24357.824} C_VEL
LIN {X 0,Y 521.156,Z 316.493,A -85,B 0,C 180,E1 24357.474,E2 24357.474} C_VEL
LIN {X 0,Y 521.816,Z 297.274,A -85,B 0,C 180,E1 24356.065,E2 24356.065} C_VEL
LIN {X 0,Y 514.978,Z 278.961,A -85,B 0,C 180,E1 24354.059,E2 24354.059} C_VEL
LIN {X 0,Y 512.679,Z 272.854,A -85,B 0,C 180,E1 24353.268,E2 24353.268} C_VEL
LIN {X 0,Y 512.623,Z 272.631,A -85,B 0,C 180,E1 24349.87,E2 24349.87} C_VEL
LIN {X 0,Y 512.61,Z 272.633,A -85,B 0,C 180,E1 24346.33,E2 24346.33} C_VEL
LIN {X 0,Y 512.639,Z 272.631,A -85,B 0,C 180,E1 24342.898,E2 24342.898} C_VEL
LIN {X 0,Y 512.649,Z 272.63,A -85,B 0,C 180,E1 24339.434,E2 24339.434} C_VEL
LIN {X 0,Y 512.604,Z 272.635,A -85,B 0,C 180,E1 24336.09,E2 24336.09} C_VEL
LIN {X 0,Y 512.644,Z 272.869,A -85,B 0,C 180,E1 24334.546,E2 24334.546} C_VEL
LIN {X 0,Y 516.614,Z 283.424,A -85,B 0,C 180,E1 24333.066,E2 24333.066} C_VEL
LIN {X 0,Y 520.776,Z 295.802,A -85,B 0,C 180,E1 24331.546,E2 24331.546} C_VEL
LIN {X 0,Y 518.7,Z 337.157,A -85,B 0,C 180,E1 24327.931,E2 24327.931} C_VEL
LIN {X 0,Y 518.616,Z 342.587,A -85,B 0,C 180,E1 24327.511,E2 24327.511} C_VEL
LIN {X 0,Y 520.868,Z 357.617,A -85,B 0,C 180,E1 24327.105,E2 24327.105} C_VEL
LIN {X 0,Y 518.908,Z 559.958,A -85,B 0,C 180,E1 24324.114,E2 24324.114} C_VEL
LIN {X 0,Y 518.407,Z 579.62,A -85,B 0,C 180,E1 24323.614,E2 24323.614} C_VEL
LIN {X 0,Y 517.798,Z 597.604,A -85,B 0,C 180,E1 24322.958,E2 24322.958} C_VEL
LIN {X 0,Y 517.068,Z 615.514,A -85,B 0,C 180,E1 24322.092,E2 24322.092} C_VEL
LIN {X 0,Y 516.22,Z 633.368,A -85,B 0,C 180,E1 24320.997,E2 24320.997} C_VEL
LIN {X 0,Y 515.38,Z 650.152,A -85,B 0,C 180,E1 24319.728,E2 24319.728} C_VEL
LIN {X 0,Y 514.552,Z 665.731,A -85,B 0,C 180,E1 24318.289,E2 24318.289} C_VEL
LIN {X 0,Y 513.83,Z 679.746,A -85,B 0,C 180,E1 24316.737,E2 24316.737} C_VEL
LIN {X 0,Y 513.204,Z 692.76,A -85,B 0,C 180,E1 24315.017,E2 24315.017} C_VEL
LIN {X 0,Y 512.71,Z 704.206,A -85,B 0,C 180,E1 24313.189,E2 24313.189} C_VEL
LIN {X 0,Y 512.352,Z 714.139,A -85,B 0,C 180,E1 24311.253,E2 24311.253} C_VEL
LIN {X 0,Y 512.116,Z 722.573,A -85,B 0,C 180,E1 24309.212,E2 24309.212} C_VEL
LIN {X 0,Y 511.992,Z 729.132,A -85,B 0,C 180,E1 24307.179,E2 24307.179} C_VEL
LIN {X 0,Y 511.937,Z 734.158,A -85,B 0,C 180,E1 24305.042,E2 24305.042} C_VEL
LIN {X 0,Y 511.914,Z 737.334,A -85,B 0,C 180,E1 24302.91,E2 24302.91} C_VEL
LIN {X 0,Y 511.917,Z 738.827,A -85,B 0,C 180,E1 24300.783,E2 24300.783} C_VEL
LIN {X 0,Y 511.911,Z 738.673,A -85,B 0,C 180,E1 24298.657,E2 24298.657} C_VEL
LIN {X 0,Y 511.912,Z 736.707,A -85,B 0,C 180,E1 24296.453,E2 24296.453} C_VEL
LIN {X 0,Y 511.942,Z 732.933,A -85,B 0,C 180,E1 24294.283,E2 24294.283} C_VEL
LIN {X 0,Y 512.015,Z 727.399,A -85,B 0,C 180,E1 24292.143,E2 24292.143} C_VEL
LIN {X 0,Y 512.174,Z 720.364,A -85,B 0,C 180,E1 24290.108,E2 24290.108} C_VEL
LIN {X 0,Y 512.432,Z 711.904,A -85,B 0,C 180,E1 24288.177,E2 24288.177} C_VEL
LIN {X 0,Y 512.822,Z 701.375,A -85,B 0,C 180,E1 24286.239,E2 24286.239} C_VEL
LIN {X 0,Y 513.355,Z 689.287,A -85,B 0,C 180,E1 24284.408,E2 24284.408} C_VEL
LIN {X 0,Y 514.033,Z 675.591,A -85,B 0,C 180,E1 24282.686,E2 24282.686} C_VEL
LIN {X 0,Y 514.776,Z 661.344,A -85,B 0,C 180,E1 24281.19,E2 24281.19} C_VEL
LIN {X 0,Y 515.609,Z 645.529,A -85,B 0,C 180,E1 24279.807,E2 24279.807} C_VEL
LIN {X 0,Y 516.449,Z 628.721,A -85,B 0,C 180,E1 24278.602,E2 24278.602} C_VEL
LIN {X 0,Y 517.278,Z 610.536,A -85,B 0,C 180,E1 24277.557,E2 24277.557} C_VEL
LIN {X 0,Y 518.022,Z 591.934,A -85,B 0,C 180,E1 24276.723,E2 24276.723} C_VEL
LIN {X 0,Y 518.599,Z 572.89,A -85,B 0,C 180,E1 24276.099,E2 24276.099} C_VEL
LIN {X 0,Y 519.014,Z 553.054,A -85,B 0,C 180,E1 24275.674,E2 24275.674} C_VEL
LIN {X 0,Y 520.123,Z 426.027,A -85,B 0,C 180,E1 24273.823,E2 24273.823} C_VEL
LIN {X 0,Y 519.314,Z 418.442,A -85,B 0,C 180,E1 24273.663,E2 24273.663} C_VEL
LIN {X 0,Y 513.976,Z 398.623,A -85,B 0,C 180,E1 24273.053,E2 24273.053} C_VEL
LIN {X 0,Y 513.364,Z 392.104,A -85,B 0,C 180,E1 24272.916,E2 24272.916} C_VEL
LIN {X 0,Y 513.545,Z 356.301,A -85,B 0,C 180,E1 24272.367,E2 24272.367} C_VEL
LIN {X 0,Y 511.161,Z 341.819,A -85,B 0,C 180,E1 24271.953,E2 24271.953} C_VEL
LIN {X 0,Y 513.119,Z 299.865,A -85,B 0,C 180,E1 24268.321,E2 24268.321} C_VEL
LIN {X 0,Y 513.068,Z 297.719,A -85,B 0,C 180,E1 24268.121,E2 24268.121} C_VEL
LIN {X 0,Y 506.338,Z 278.626,A -85,B 0,C 180,E1 24265.833,E2 24265.833} C_VEL
LIN {X 0,Y 504.722,Z 273.804,A -85,B 0,C 180,E1 24265.195,E2 24265.195} C_VEL
LIN {X 0,Y 504.673,Z 273.62,A -85,B 0,C 180,E1 24261.819,E2 24261.819} C_VEL
LIN {X 0,Y 504.694,Z 273.612,A -85,B 0,C 180,E1 24258.322,E2 24258.322} C_VEL
LIN {X 0,Y 504.706,Z 273.617,A -85,B 0,C 180,E1 24254.827,E2 24254.827} C_VEL
LIN {X 0,Y 504.71,Z 273.619,A -85,B 0,C 180,E1 24251.277,E2 24251.277} C_VEL
LIN {X 0,Y 504.699,Z 273.618,A -85,B 0,C 180,E1 24247.747,E2 24247.747} C_VEL
LIN {X 0,Y 504.707,Z 273.613,A -85,B 0,C 180,E1 24244.238,E2 24244.238} C_VEL
LIN {X 0,Y 504.69,Z 273.612,A -85,B 0,C 180,E1 24240.703,E2 24240.703} C_VEL
LIN {X 0,Y 504.681,Z 273.619,A -85,B 0,C 180,E1 24237.183,E2 24237.183} C_VEL
LIN {X 0,Y 504.705,Z 273.616,A -85,B 0,C 180,E1 24233.714,E2 24233.714} C_VEL
LIN {X 0,Y 504.708,Z 273.614,A -85,B 0,C 180,E1 24230.165,E2 24230.165} C_VEL
LIN {X 0,Y 504.659,Z 273.622,A -85,B 0,C 180,E1 24226.815,E2 24226.815} C_VEL
LIN {X 0,Y 504.648,Z 273.601,A -85,B 0,C 180,E1 24223.288,E2 24223.288} C_VEL
LIN {X 0,Y 504.657,Z 273.717,A -85,B 0,C 180,E1 24220.792,E2 24220.792} C_VEL
LIN {X 0,Y 505.095,Z 275.399,A -85,B 0,C 180,E1 24220.552,E2 24220.552} C_VEL
LIN {X 0,Y 511.329,Z 294.509,A -85,B 0,C 180,E1 24218.576,E2 24218.576} C_VEL
LIN {X 0,Y 510.714,Z 334.383,A -85,B 0,C 180,E1 24215.337,E2 24215.337} C_VEL
LIN {X 0,Y 509.833,Z 376.612,A -85,B 0,C 180,E1 24211.912,E2 24211.912} C_VEL
LIN {X 0,Y 508.721,Z 421.729,A -85,B 0,C 180,E1 24208.256,E2 24208.256} C_VEL
LIN {X 0,Y 507.706,Z 464.389,A -85,B 0,C 180,E1 24204.804,E2 24204.804} C_VEL
LIN {X 0,Y 507.513,Z 474.435,A -85,B 0,C 180,E1 24204.018,E2 24204.018} C_VEL
LIN {X 0,Y 508.534,Z 485.17,A -85,B 0,C 180,E1 24203.818,E2 24203.818} C_VEL
LIN {X 0,Y 507.591,Z 616.922,A -85,B 0,C 180,E1 24201.898,E2 24201.898} C_VEL
LIN {X 0,Y 507.323,Z 632.874,A -85,B 0,C 180,E1 24201.458,E2 24201.458} C_VEL
LIN {X 0,Y 506.925,Z 648.572,A -85,B 0,C 180,E1 24200.808,E2 24200.808} C_VEL
LIN {X 0,Y 506.455,Z 663.014,A -85,B 0,C 180,E1 24199.997,E2 24199.997} C_VEL
LIN {X 0,Y 505.905,Z 677.326,A -85,B 0,C 180,E1 24198.949,E2 24198.949} C_VEL
LIN {X 0,Y 505.414,Z 690.119,A -85,B 0,C 180,E1 24197.766,E2 24197.766} C_VEL
LIN {X 0,Y 504.93,Z 702.107,A -85,B 0,C 180,E1 24196.372,E2 24196.372} C_VEL
LIN {X 0,Y 504.569,Z 711.921,A -85,B 0,C 180,E1 24194.956,E2 24194.956} C_VEL
LIN {X 0,Y 504.268,Z 721.08,A -85,B 0,C 180,E1 24193.276,E2 24193.276} C_VEL
LIN {X 0,Y 504.091,Z 728.094,A -85,B 0,C 180,E1 24191.618,E2 24191.618} C_VEL
LIN {X 0,Y 503.989,Z 733.734,A -85,B 0,C 180,E1 24189.783,E2 24189.783} C_VEL
LIN {X 0,Y 503.95,Z 737.461,A -85,B 0,C 180,E1 24187.978,E2 24187.978} C_VEL
LIN {X 0,Y 503.935,Z 739.424,A -85,B 0,C 180,E1 24186.126,E2 24186.126} C_VEL
LIN {X 0,Y 503.935,Z 739.676,A -85,B 0,C 180,E1 24184.247,E2 24184.247} C_VEL
LIN {X 0,Y 503.943,Z 738.029,A -85,B 0,C 180,E1 24182.339,E2 24182.339} C_VEL
LIN {X 0,Y 503.976,Z 734.754,A -85,B 0,C 180,E1 24180.529,E2 24180.529} C_VEL
LIN {X 0,Y 504.057,Z 729.721,A -85,B 0,C 180,E1 24178.754,E2 24178.754} C_VEL
LIN {X 0,Y 504.23,Z 722.652,A -85,B 0,C 180,E1 24176.956,E2 24176.956} C_VEL
LIN {X 0,Y 504.492,Z 714.234,A -85,B 0,C 180,E1 24175.335,E2 24175.335} C_VEL
LIN {X 0,Y 504.853,Z 704.388,A -85,B 0,C 180,E1 24173.832,E2 24173.832} C_VEL
LIN {X 0,Y 505.3,Z 693.074,A -85,B 0,C 180,E1 24172.452,E2 24172.452} C_VEL
LIN {X 0,Y 505.831,Z 679.711,A -85,B 0,C 180,E1 24171.152,E2 24171.152} C_VEL
LIN {X 0,Y 506.327,Z 666.781,A -85,B 0,C 180,E1 24170.158,E2 24170.158} C_VEL
LIN {X 0,Y 506.852,Z 651.387,A -85,B 0,C 180,E1 24169.237,E2 24169.237} C_VEL
LIN {X 0,Y 507.266,Z 635.918,A -85,B 0,C 180,E1 24168.558,E2 24168.558} C_VEL
LIN {X 0,Y 507.556,Z 619.27,A -85,B 0,C 180,E1 24168.06,E2 24168.06} C_VEL
LIN {X 0,Y 507.753,Z 593.359,A -85,B 0,C 180,E1 24167.644,E2 24167.644} C_VEL
LIN {X 0,Y 508.34,Z 481.293,A -85,B 0,C 180,E1 24166.026,E2 24166.026} C_VEL
LIN {X 0,Y 507.457,Z 474.005,A -85,B 0,C 180,E1 24165.865,E2 24165.865} C_VEL
LIN {X 0,Y 508.502,Z 429.195,A -85,B 0,C 180,E1 24162.259,E2 24162.259} C_VEL
LIN {X 0,Y 509.471,Z 389.356,A -85,B 0,C 180,E1 24159.049,E2 24159.049} C_VEL
LIN {X 0,Y 510.24,Z 346.659,A -85,B 0,C 180,E1 24155.654,E2 24155.654} C_VEL
LIN {X 0,Y 510.701,Z 309.068,A -85,B 0,C 180,E1 24152.666,E2 24152.666} C_VEL
LIN {X 0,Y 510.741,Z 292.979,A -85,B 0,C 180,E1 24151.382,E2 24151.382} C_VEL
LIN {X 0,Y 504.771,Z 274.004,A -85,B 0,C 180,E1 24149.488,E2 24149.488} C_VEL
LIN {X 0,Y 504.69,Z 273.619,A -85,B 0,C 180,E1 24149.115,E2 24149.115} C_VEL
LIN {X 0,Y 504.709,Z 273.616,A -85,B 0,C 180,E1 24145.664,E2 24145.664} C_VEL
LIN {X 0,Y 504.669,Z 273.622,A -85,B 0,C 180,E1 24142.236,E2 24142.236} C_VEL
LIN {X 0,Y 504.671,Z 273.614,A -85,B 0,C 180,E1 24138.721,E2 24138.721} C_VEL
LIN {X 0,Y 504.711,Z 273.613,A -85,B 0,C 180,E1 24135.261,E2 24135.261} C_VEL
LIN {X 0,Y 504.694,Z 273.622,A -85,B 0,C 180,E1 24131.775,E2 24131.775} C_VEL
LIN {X 0,Y 504.667,Z 273.617,A -85,B 0,C 180,E1 24128.316,E2 24128.316} C_VEL
LIN {X 0,Y 504.687,Z 273.615,A -85,B 0,C 180,E1 24124.808,E2 24124.808} C_VEL
LIN {X 0,Y 504.711,Z 273.617,A -85,B 0,C 180,E1 24121.363,E2 24121.363} C_VEL
LIN {X 0,Y 504.675,Z 273.618,A -85,B 0,C 180,E1 24117.957,E2 24117.957} C_VEL
LIN {X 0,Y 504.673,Z 273.617,A -85,B 0,C 180,E1 24114.429,E2 24114.429} C_VEL
LIN {X 0,Y 504.709,Z 273.612,A -85,B 0,C 180,E1 24110.996,E2 24110.996} C_VEL
LIN {X 0,Y 504.704,Z 273.617,A -85,B 0,C 180,E1 24107.414,E2 24107.414} C_VEL
LIN {X 0,Y 504.673,Z 273.615,A -85,B 0,C 180,E1 24104.015,E2 24104.015} C_VEL
LIN {X 0,Y 504.69,Z 273.614,A -85,B 0,C 180,E1 24100.559,E2 24100.559} C_VEL
LIN {X 0,Y 504.712,Z 273.617,A -85,B 0,C 180,E1 24097.029,E2 24097.029} C_VEL
LIN {X 0,Y 504.691,Z 273.62,A -85,B 0,C 180,E1 24093.529,E2 24093.529} C_VEL
LIN {X 0,Y 504.676,Z 273.615,A -85,B 0,C 180,E1 24090.049,E2 24090.049} C_VEL
LIN {X 0,Y 504.704,Z 273.613,A -85,B 0,C 180,E1 24086.583,E2 24086.583} C_VEL
LIN {X 0,Y 504.708,Z 273.62,A -85,B 0,C 180,E1 24083.112,E2 24083.112} C_VEL
LIN {X 0,Y 504.68,Z 273.619,A -85,B 0,C 180,E1 24079.621,E2 24079.621} C_VEL
LIN {X 0,Y 504.684,Z 273.618,A -85,B 0,C 180,E1 24076.1,E2 24076.1} C_VEL
LIN {X 0,Y 504.71,Z 273.617,A -85,B 0,C 180,E1 24072.648,E2 24072.648} C_VEL
LIN {X 0,Y 504.713,Z 273.617,A -85,B 0,C 180,E1 24069.046,E2 24069.046} C_VEL
LIN {X 0,Y 504.722,Z 273.854,A -85,B 0,C 180,E1 24067.355,E2 24067.355} C_VEL
LIN {X 0,Y 507.634,Z 281.444,A -85,B 0,C 180,E1 24066.429,E2 24066.429} C_VEL
LIN {X 0,Y 515.207,Z 300.924,A -85,B 0,C 180,E1 24064.281,E2 24064.281} C_VEL
LIN {X 0,Y 514.589,Z 316.443,A -85,B 0,C 180,E1 24063.136,E2 24063.136} C_VEL
LIN {X 0,Y 517.105,Z 333.218,A -85,B 0,C 180,E1 24062.679,E2 24062.679} C_VEL
LIN {X 0,Y 514.727,Z 530.291,A -85,B 0,C 180,E1 24059.668,E2 24059.668} C_VEL
LIN {X 0,Y 514.183,Z 578.441,A -85,B 0,C 180,E1 24058.929,E2 24058.929} C_VEL
LIN {X 0,Y 513.538,Z 599.827,A -85,B 0,C 180,E1 24058.392,E2 24058.392} C_VEL
LIN {X 0,Y 512.738,Z 620.455,A -85,B 0,C 180,E1 24057.651,E2 24057.651} C_VEL
LIN {X 0,Y 511.825,Z 639.514,A -85,B 0,C 180,E1 24056.76,E2 24056.76} C_VEL
LIN {X 0,Y 510.774,Z 658.935,A -85,B 0,C 180,E1 24055.632,E2 24055.632} C_VEL
LIN {X 0,Y 509.701,Z 677.368,A -85,B 0,C 180,E1 24054.326,E2 24054.326} C_VEL
LIN {X 0,Y 508.649,Z 693.186,A -85,B 0,C 180,E1 24052.965,E2 24052.965} C_VEL
LIN {X 0,Y 507.519,Z 709.709,A -85,B 0,C 180,E1 24051.275,E2 24051.275} C_VEL
LIN {X 0,Y 506.541,Z 724.454,A -85,B 0,C 180,E1 24049.485,E2 24049.485} C_VEL
LIN {X 0,Y 505.731,Z 737.586,A -85,B 0,C 180,E1 24047.606,E2 24047.606} C_VEL
LIN {X 0,Y 505.077,Z 749.383,A -85,B 0,C 180,E1 24045.617,E2 24045.617} C_VEL
LIN {X 0,Y 504.568,Z 760.338,A -85,B 0,C 180,E1 24043.404,E2 24043.404} C_VEL
LIN {X 0,Y 504.236,Z 769.256,A -85,B 0,C 180,E1 24041.204,E2 24041.204} C_VEL
LIN {X 0,Y 504.048,Z 776.587,A -85,B 0,C 180,E1 24038.938,E2 24038.938} C_VEL
LIN {X 0,Y 503.957,Z 782.261,A -85,B 0,C 180,E1 24036.606,E2 24036.606} C_VEL
LIN {X 0,Y 503.916,Z 786.089,A -85,B 0,C 180,E1 24034.323,E2 24034.323} C_VEL
LIN {X 0,Y 503.911,Z 788.374,A -85,B 0,C 180,E1 24031.932,E2 24031.932} C_VEL
LIN {X 0,Y 503.9,Z 788.917,A -85,B 0,C 180,E1 24029.544,E2 24029.544} C_VEL
LIN {X 0,Y 503.911,Z 787.842,A -85,B 0,C 180,E1 24027.269,E2 24027.269} C_VEL
LIN {X 0,Y 503.922,Z 785.126,A -85,B 0,C 180,E1 24024.99,E2 24024.99} C_VEL
LIN {X 0,Y 503.964,Z 780.733,A -85,B 0,C 180,E1 24022.704,E2 24022.704} C_VEL
LIN {X 0,Y 504.091,Z 774.616,A -85,B 0,C 180,E1 24020.408,E2 24020.408} C_VEL
LIN {X 0,Y 504.314,Z 767.088,A -85,B 0,C 180,E1 24018.216,E2 24018.216} C_VEL
LIN {X 0,Y 504.683,Z 757.701,A -85,B 0,C 180,E1 24016.012,E2 24016.012} C_VEL
LIN {X 0,Y 505.219,Z 746.825,A -85,B 0,C 180,E1 24013.914,E2 24013.914} C_VEL
LIN {X 0,Y 505.915,Z 734.462,A -85,B 0,C 180,E1 24011.918,E2 24011.918} C_VEL
LIN {X 0,Y 506.779,Z 720.73,A -85,B 0,C 180,E1 24010.041,E2 24010.041} C_VEL
LIN {X 0,Y 507.8,Z 705.486,A -85,B 0,C 180,E1 24008.273,E2 24008.273} C_VEL
LIN {X 0,Y 508.908,Z 689.266,A -85,B 0,C 180,E1 24006.678,E2 24006.678} C_VEL
LIN {X 0,Y 509.9,Z 674.301,A -85,B 0,C 180,E1 24005.435,E2 24005.435} C_VEL
LIN {X 0,Y 510.85,Z 656.652,A -85,B 0,C 180,E1 24004.245,E2 24004.245} C_VEL
LIN {X 0,Y 511.789,Z 637.288,A -85,B 0,C 180,E1 24003.172,E2 24003.172} C_VEL
LIN {X 0,Y 512.652,Z 616.924,A -85,B 0,C 180,E1 24002.278,E2 24002.278} C_VEL
LIN {X 0,Y 513.334,Z 596.303,A -85,B 0,C 180,E1 24001.594,E2 24001.594} C_VEL
LIN {X 0,Y 513.865,Z 575.457,A -85,B 0,C 180,E1 24001.112,E2 24001.112} C_VEL
LIN {X 0,Y 515.691,Z 379.054,A -85,B 0,C 180,E1 23998.21,E2 23998.21} C_VEL
LIN {X 0,Y 516.094,Z 330.597,A -85,B 0,C 180,E1 23997.438,E2 23997.438} C_VEL
LIN {X 0,Y 513.987,Z 317.144,A -85,B 0,C 180,E1 23997.062,E2 23997.062} C_VEL
LIN {X 0,Y 514.567,Z 300.018,A -85,B 0,C 180,E1 23995.77,E2 23995.77} C_VEL
LIN {X 0,Y 508.155,Z 282.576,A -85,B 0,C 180,E1 23993.777,E2 23993.777} C_VEL
LIN {X 0,Y 504.746,Z 274.031,A -85,B 0,C 180,E1 23992.624,E2 23992.624} C_VEL
LIN {X 0,Y 504.688,Z 273.622,A -85,B 0,C 180,E1 23991.861,E2 23991.861} C_VEL
LIN {X 0,Y 504.673,Z 273.623,A -85,B 0,C 180,E1 23988.323,E2 23988.323} C_VEL
LIN {X 0,Y 504.696,Z 273.622,A -85,B 0,C 180,E1 23984.826,E2 23984.826} C_VEL
LIN {X 0,Y 504.715,Z 273.618,A -85,B 0,C 180,E1 23981.276,E2 23981.276} C_VEL
LIN {X 0,Y 504.672,Z 273.622,A -85,B 0,C 180,E1 23977.892,E2 23977.892} C_VEL
LIN {X 0,Y 504.745,Z 273.87,A -85,B 0,C 180,E1 23975.27,E2 23975.27} C_VEL
LIN {X 0,Y 509.029,Z 284.919,A -85,B 0,C 180,E1 23973.607,E2 23973.607} C_VEL
LIN {X 0,Y 513.704,Z 298.842,A -85,B 0,C 180,E1 23971.818,E2 23971.818} C_VEL
LIN {X 0,Y 511.459,Z 339.199,A -85,B 0,C 180,E1 23968.235,E2 23968.235} C_VEL
LIN {X 0,Y 511.524,Z 342.462,A -85,B 0,C 180,E1 23968.013,E2 23968.013} C_VEL
LIN {X 0,Y 513.978,Z 358.746,A -85,B 0,C 180,E1 23967.544,E2 23967.544} C_VEL
LIN {X 0,Y 512.461,Z 472.725,A -85,B 0,C 180,E1 23965.787,E2 23965.787} C_VEL
LIN {X 0,Y 511.596,Z 560.324,A -85,B 0,C 180,E1 23964.472,E2 23964.472} C_VEL
LIN {X 0,Y 511.05,Z 580.056,A -85,B 0,C 180,E1 23963.961,E2 23963.961} C_VEL
LIN {X 0,Y 510.37,Z 598.506,A -85,B 0,C 180,E1 23963.273,E2 23963.273} C_VEL
LIN {X 0,Y 509.549,Z 616.547,A -85,B 0,C 180,E1 23962.375,E2 23962.375} C_VEL
LIN {X 0,Y 508.634,Z 634.223,A -85,B 0,C 180,E1 23961.265,E2 23961.265} C_VEL
LIN {X 0,Y 507.715,Z 650.838,A -85,B 0,C 180,E1 23959.979,E2 23959.979} C_VEL
LIN {X 0,Y 506.811,Z 666.298,A -85,B 0,C 180,E1 23958.519,E2 23958.519} C_VEL
LIN {X 0,Y 505.995,Z 680.673,A -85,B 0,C 180,E1 23956.886,E2 23956.886} C_VEL
LIN {X 0,Y 505.316,Z 693.54,A -85,B 0,C 180,E1 23955.14,E2 23955.14} C_VEL
LIN {X 0,Y 504.78,Z 704.869,A -85,B 0,C 180,E1 23953.283,E2 23953.283} C_VEL
LIN {X 0,Y 504.389,Z 714.671,A -85,B 0,C 180,E1 23951.317,E2 23951.317} C_VEL
LIN {X 0,Y 504.132,Z 722.981,A -85,B 0,C 180,E1 23949.244,E2 23949.244} C_VEL
LIN {X 0,Y 503.996,Z 729.437,A -85,B 0,C 180,E1 23947.179,E2 23947.179} C_VEL
LIN {X 0,Y 503.938,Z 734.369,A -85,B 0,C 180,E1 23945.008,E2 23945.008} C_VEL
LIN {X 0,Y 503.913,Z 737.461,A -85,B 0,C 180,E1 23942.843,E2 23942.843} C_VEL
LIN {X 0,Y 503.914,Z 738.851,A -85,B 0,C 180,E1 23940.682,E2 23940.682} C_VEL
LIN {X 0,Y 503.911,Z 738.608,A -85,B 0,C 180,E1 23938.522,E2 23938.522} C_VEL
LIN {X 0,Y 503.912,Z 736.66,A -85,B 0,C 180,E1 23936.359,E2 23936.359} C_VEL
LIN {X 0,Y 503.945,Z 732.928,A -85,B 0,C 180,E1 23934.192,E2 23934.192} C_VEL
LIN {X 0,Y 504.03,Z 727.395,A -85,B 0,C 180,E1 23932.018,E2 23932.018} C_VEL
LIN {X 0,Y 504.204,Z 720.361,A -85,B 0,C 180,E1 23929.95,E2 23929.95} C_VEL
LIN {X 0,Y 504.494,Z 711.898,A -85,B 0,C 180,E1 23927.989,E2 23927.989} C_VEL
LIN {X 0,Y 504.931,Z 701.366,A -85,B 0,C 180,E1 23926.02,E2 23926.02} C_VEL
LIN {X 0,Y 505.526,Z 689.278,A -85,B 0,C 180,E1 23924.16,E2 23924.16} C_VEL
LIN {X 0,Y 506.277,Z 675.582,A -85,B 0,C 180,E1 23922.412,E2 23922.412} C_VEL
LIN {X 0,Y 507.096,Z 661.337,A -85,B 0,C 180,E1 23920.894,E2 23920.894} C_VEL
LIN {X 0,Y 508.011,Z 645.517,A -85,B 0,C 180,E1 23919.492,E2 23919.492} C_VEL
LIN {X 0,Y 508.934,Z 628.612,A -85,B 0,C 180,E1 23918.264,E2 23918.264} C_VEL
LIN {X 0,Y 509.832,Z 610.521,A -85,B 0,C 180,E1 23917.211,E2 23917.211} C_VEL
LIN {X 0,Y 510.615,Z 592.575,A -85,B 0,C 180,E1 23916.394,E2 23916.394} C_VEL
LIN {X 0,Y 511.25,Z 573.74,A -85,B 0,C 180,E1 23915.758,E2 23915.758} C_VEL
LIN {X 0,Y 511.696,Z 554.425,A -85,B 0,C 180,E1 23915.329,E2 23915.329} C_VEL
LIN {X 0,Y 513.364,Z 392.104,A -85,B 0,C 180,E1 23912.916,E2 23912.916} C_VEL
LIN {X 0,Y 512.593,Z 383.441,A -85,B 0,C 180,E1 23912.736,E2 23912.736} C_VEL
LIN {X 0,Y 506.641,Z 358.228,A -85,B 0,C 180,E1 23911.968,E2 23911.968} C_VEL
LIN {X 0,Y 503.93,Z 341.479,A -85,B 0,C 180,E1 23911.47,E2 23911.47} C_VEL
